// TwinCAT 3 PLC project lcls_plc_dream_vac
// ProgramVersion: 3.1.4022.7
// libraries:
//   LCLS General, * (SLAC)
//   LCLS Vacuum, * (SLAC - LCLS)
//   LCLSVacuumSerialDriverLib, * (SLAC - LCLS)
//   PMPS, * (SLAC - LCLS)
//   Tc2_SerialCom, * (Beckhoff Automation GmbH)
//   Tc2_Standard, * (Beckhoff Automation GmbH)
//   Tc2_System, * (Beckhoff Automation GmbH)
//   Tc3_Module, * (Beckhoff Automation GmbH)
// project tree:
//   DUTs/ E_Op.TcDUT, E_OpStep.TcDUT
//   GVLs/ GVL_Automation.TcGVL, GVL_Constants.TcGVL, GVL_FWM.TcGVL, GVL_PLC_Interface.TcGVL, GVL_Serial_Com.TcGVL, GVL_TC.TcGVL, GVL_VAC_GAUGES.TcGVL, GVL_VAC_PUMPS.TcGVL, GVL_VAC_VALVES.TcGVL, GVL_Variables.TcGVL
//   / PlcTask.TcTTO, Serial_COM.TcTTO
//   POUs/Automation/Abstracts/ FB_Operation.TcPOU
//   POUs/Automation/ FB_VentMcCat.TcPOU, FB_AtVacuum.TcPOU
//   POUs/Functions/ F_AllPumpsRunning.TcPOU, F_IsValidStateTransition.TcPOU, F_PressAtVacSP.TcPOU, F_TurboIlkLogic.TcPOU
//   POUs/ PRG_AUTOMATION.TcPOU, MAIN.TcPOU, PRG_COM.TcPOU, PRG_ECAT_CHECK.TcPOU, PRG_GAUGES.TcPOU, PRG_HV_ILK.TcPOU, PRG_COIL_PS_ILK.TcPOU, PRG_TC.TcPOU, PRG_TURBO_PUMPS.TcPOU, PRG_VALVES.TcPOU
// real-time tasks:
//   TASK PlcTask: cycle T#10ms, priority 20, ADS port 350
//   TASK Serial_COM: cycle T#2ms, priority 19, ADS port 351
// I/O:
//   DEVICE Device 1 (EtherCAT), AmsNetId 172.21.132.159.2.1
//     R20_DRL_03_CX0_EK1200 [EK1200-5000 EtherCAT Power supply (2A E-Bus)]
//       R20_DRL_03_E1_EL2202
//       R20_DRL_03_E2_EL6070 [EL6070 1Ch. Licensing-Terminal]
//       R20_DRL_03_E3_EL9070 [EL9070 Shield terminal]
//       R20_DRL_03_E4_EL1004 [EL1004 4Ch. Dig. Input 24V, 3ms]
//       R20_DRL_03_E5_EL1004 [EL1004 4Ch. Dig. Input 24V, 3ms]
//       R20_DRL_03_E6_EL1004
//       R20_DRL_03_E7_EL2794 [EL2794 4Ch. Dig. Output 24V AC/DC, 2A, short-circuit-proof]
//       R20_DRL_03_E8_EL2794 [EL2794 4Ch. Dig. Output 24V AC/DC, 2A, short-circuit-proof]
//       R20_DRL_03_E9_EL6001 [EL6001 Interface (RS232)]
//       R20_DRL_03_E10_EL6001 [EL6001 Interface (RS232)]
//       R20_DRL_03_E11_EL6001 [EL6001 Interface (RS232)]
//       R20_DRL_03_E12_EL6001 [EL6001 Interface (RS232)]
//       R20_DRL_03_E13_EL9505 [EL9505 Power supply terminal 5V]
//       R20_DRL_03_E14_EL6695 [EL6695 EtherCAT Bridge terminal (Primary)]
//       R20_DRL_03_E15_EL1122 [EK1122 2 port EtherCAT junction]
//         K4S8_DRL_03_EK0_EK1100 [EK1100 EtherCAT Coupler (2A E-Bus)]
//           K4S8_DRL_03_E1_EL2624 [EL2624 4Ch. Relay Output, NO (125V AC / 30V DC)]
//           K4S8_DRL_03_E2_EL9184 [EL9184 Potential Connection, 8 x 24V, 8 x Ground]
//           K4S8_DRL_03_E3_EL9070 [EL9070 Shield terminal]
//           K4S8_DRL_03_E4_EL1084 [EL1084 4Ch. Dig. Input 24V, 3ms, negative]
//           K4S8_DRL_03_E5_EL3174-0002 [EL3174-0002 4Ch. Ana. Input +/-10V, +/-20mA 16 Bit, Isolated Channels]
//           K4S8_DRL_03_E6_EL3174-0002 [EL3174-0002 4Ch. Ana. Input +/-10V, +/-20mA 16 Bit, Isolated Channels]
//           K4S8_DRL_03_E7_EL9505 [EL9505 Power supply terminal 5V]
//           K4S8_DRL_03_E8_EL1124 [EL1124 4Ch. Dig. Input 5V, 10µs, Sensor Power]
//           K4S8_DRL_03_E9_EL9410 [EL9410 E-Bus Power Supplier  (Diagnostics)]
//           K4S8_DRL_03_E10_EL1004 [EL1004 4Ch. Dig. Input 24V, 3ms]
//           K4S8_DRL_03_E11_EL2004 [EL2004 4Ch. Dig. Output 24V, 0.5A]
//           K4S8_DRL_03_E12_EL6021 [EL6021 Interface (RS422/485)]
//           K4S8_DRL_03_E13_EL1004 [EL1004 4Ch. Dig. Input 24V, 3ms]
//           K4S8_DRL_03_E14_EL2004 [EL2004 4Ch. Dig. Output 24V, 0.5A]
//           K4S8_DRL_03_E15_EL6021 [EL6021 Interface (RS422/485)]
//           K4S8_DRL_03_E16_EL1004 [EL1004 4Ch. Dig. Input 24V, 3ms]
//           K4S8_DRL_03_E17_EL2004 [EL2004 4Ch. Dig. Output 24V, 0.5A]
//           K4S8_DRL_03_E18_EL6021 [EL6021 Interface (RS422/485)]
//           K4S8_DRL_03_E19_EL1004 [EL1004 4Ch. Dig. Input 24V, 3ms]
//           K4S8_DRL_03_E20_EL2004 [EL2004 4Ch. Dig. Output 24V, 0.5A]
//           K4S8_DRL_03_E21_EL3052 [EL3052 2Ch. Ana. Input 4-20mA]
//           K4S8_DRL_03_E22_EL3314 [EL3314 4Ch. Ana. Input Thermocouple (TC)]
//           K4S8_DRL_03_E23_EL3314 [EL3314 4Ch. Ana. Input Thermocouple (TC)]
//           K4S8_DRL_03_E24_EL9011
//         K4S8_DRL_04_EK0_EK1100 [EK1100 EtherCAT Coupler (2A E-Bus)]
//           K4S8_DRL_04_E1_EL1004 [EL1004 4Ch. Dig. Input 24V, 3ms]
//           K4S8_DRL_04_E2_EL2004 [EL2004 4Ch. Dig. Output 24V, 0.5A]
//           K4S8_DRL_04_E3_EL1004 [EL1004 4Ch. Dig. Input 24V, 3ms]
//           K4S8_DRL_04_E4_EL1004 [EL1004 4Ch. Dig. Input 24V, 3ms]
//           K4S8_DRL_04_E5_EL2794 [EL2794 4Ch. Dig. Output 24V AC/DC, 2A, short-circuit-proof]
//           K4S8_DRL_04_E6_EL6001 [EL6001 Interface (RS232)]
//           K4S8_DRL_04_E7_EL6001 [EL6001 Interface (RS232)]
//           K4S8_DRL_04_E8_EL6001 [EL6001 Interface (RS232)]
//           K4S8_DRL_04_E9_EL1004 [EL1004 4Ch. Dig. Input 24V, 3ms]
//           K4S8_DRL_04_E10_EL1004 [EL1004 4Ch. Dig. Input 24V, 3ms]
//           K4S8_DRL_04_E11_EL2004
//           K4S8_DRL_04_E12_EL9184 [EL9184 Potential Connection, 8 x 24V, 8 x Ground]
//           K4S8_DRL_04_E13_EL9070 [EL9070 Shield terminal]
//           K4S8_DRL_04_E14_EL2624 [EL2624 4Ch. Relay Output, NO (125V AC / 30V DC)]
//           K4S8_DRL_04_E15_EL1084 [EL1084 4Ch. Dig. Input 24V, 3ms, negative]
//           K4S8_DRL_04_E16_EL3174-0002 [EL3174-0002 4Ch. Ana. Input +/-10V, +/-20mA 16 Bit, Isolated Channels]
//           K4S8_DRL_04_E17_EL6001 [EL6001 Interface (RS232)]
//           K4S8_DRL_04_E18_EL9011
//         K4S8_DRL_04_EP1_EP4374-0002 [EP4374-0002 2Ch. Ana. Input +/-10V, 0-10V, 0/4-20mA configurable; 2Ch. Ana. Output +/-10V, 0-10V, 0/4-20mA configurable]
//         K4S8_DRL_04_EP2_EP4374-0002 [EP4374-0002 2Ch. Ana. Input +/-10V, 0-10V, 0/4-20mA configurable; 2Ch. Ana. Output +/-10V, 0-10V, 0/4-20mA configurable]
//         R03_DRL_01_EK1100 [EK1100 EtherCAT Coupler (2A E-Bus)]
//           R03_DRL_01_E1_EL1004 [EL1004 4Ch. Dig. Input 24V, 3ms]
//           R03_DRL_01_E2_EL2624 [EL2624 4Ch. Relay Output, NO (125V AC / 30V DC)]
//           R03_DRL_01_E3_EL3174-0002 [EL3174-0002 4Ch. Ana. Input +/-10V, +/-20mA 16 Bit, Isolated Channels]
//           R03_DRL_01_E4_EK1110 [EK1110 EtherCAT extension]
//         WALL_E_PPL_01_EP1_EP4374-0002 [EP4374-0002 2Ch. Ana. Input +/-10V, 0-10V, 0/4-20mA configurable; 2Ch. Ana. Output +/-10V, 0-10V, 0/4-20mA configurable]
//         WALL_E_PPL_01_EP2_EP2338-0002 [EP2338-0002 8 Ch. Dig. Input/Output 24V, 0,5A, M12]
// variable links:
//   lcls_plc_dream_vac Instance <-> Device 1 (EtherCAT)/R20_DRL_03_CX0_EK1200/R20_DRL_03_E10_EL6001
//     Serial_COM Inputs/GVL_Serial_Com.stComIn_DREAM_DP3_PTM_01/D[0] <-> COM Inputs/Data In 0
//     Serial_COM Inputs/GVL_Serial_Com.stComIn_DREAM_DP3_PTM_01/D[10] <-> COM Inputs/Data In 10
//     Serial_COM Inputs/GVL_Serial_Com.stComIn_DREAM_DP3_PTM_01/D[11] <-> COM Inputs/Data In 11
//     Serial_COM Inputs/GVL_Serial_Com.stComIn_DREAM_DP3_PTM_01/D[12] <-> COM Inputs/Data In 12
//     Serial_COM Inputs/GVL_Serial_Com.stComIn_DREAM_DP3_PTM_01/D[13] <-> COM Inputs/Data In 13
//     Serial_COM Inputs/GVL_Serial_Com.stComIn_DREAM_DP3_PTM_01/D[14] <-> COM Inputs/Data In 14
//     Serial_COM Inputs/GVL_Serial_Com.stComIn_DREAM_DP3_PTM_01/D[15] <-> COM Inputs/Data In 15
//     Serial_COM Inputs/GVL_Serial_Com.stComIn_DREAM_DP3_PTM_01/D[16] <-> COM Inputs/Data In 16
//     Serial_COM Inputs/GVL_Serial_Com.stComIn_DREAM_DP3_PTM_01/D[17] <-> COM Inputs/Data In 17
//     Serial_COM Inputs/GVL_Serial_Com.stComIn_DREAM_DP3_PTM_01/D[18] <-> COM Inputs/Data In 18
//     Serial_COM Inputs/GVL_Serial_Com.stComIn_DREAM_DP3_PTM_01/D[19] <-> COM Inputs/Data In 19
//     Serial_COM Inputs/GVL_Serial_Com.stComIn_DREAM_DP3_PTM_01/D[1] <-> COM Inputs/Data In 1
//     Serial_COM Inputs/GVL_Serial_Com.stComIn_DREAM_DP3_PTM_01/D[20] <-> COM Inputs/Data In 20
//     Serial_COM Inputs/GVL_Serial_Com.stComIn_DREAM_DP3_PTM_01/D[21] <-> COM Inputs/Data In 21
//     Serial_COM Inputs/GVL_Serial_Com.stComIn_DREAM_DP3_PTM_01/D[2] <-> COM Inputs/Data In 2
//     Serial_COM Inputs/GVL_Serial_Com.stComIn_DREAM_DP3_PTM_01/D[3] <-> COM Inputs/Data In 3
//     Serial_COM Inputs/GVL_Serial_Com.stComIn_DREAM_DP3_PTM_01/D[4] <-> COM Inputs/Data In 4
//     Serial_COM Inputs/GVL_Serial_Com.stComIn_DREAM_DP3_PTM_01/D[5] <-> COM Inputs/Data In 5
//     Serial_COM Inputs/GVL_Serial_Com.stComIn_DREAM_DP3_PTM_01/D[6] <-> COM Inputs/Data In 6
//     Serial_COM Inputs/GVL_Serial_Com.stComIn_DREAM_DP3_PTM_01/D[7] <-> COM Inputs/Data In 7
//     Serial_COM Inputs/GVL_Serial_Com.stComIn_DREAM_DP3_PTM_01/D[8] <-> COM Inputs/Data In 8
//     Serial_COM Inputs/GVL_Serial_Com.stComIn_DREAM_DP3_PTM_01/D[9] <-> COM Inputs/Data In 9
//     Serial_COM Inputs/GVL_Serial_Com.stComIn_DREAM_DP3_PTM_01/Status <-> COM Inputs/Status
//     Serial_COM Outputs/GVL_Serial_Com.stComOut_DREAM_DP3_PTM_01/Ctrl <-> COM Outputs/Ctrl
//     Serial_COM Outputs/GVL_Serial_Com.stComOut_DREAM_DP3_PTM_01/D[0] <-> COM Outputs/Data Out 0
//     Serial_COM Outputs/GVL_Serial_Com.stComOut_DREAM_DP3_PTM_01/D[10] <-> COM Outputs/Data Out 10
//     Serial_COM Outputs/GVL_Serial_Com.stComOut_DREAM_DP3_PTM_01/D[11] <-> COM Outputs/Data Out 11
//     Serial_COM Outputs/GVL_Serial_Com.stComOut_DREAM_DP3_PTM_01/D[12] <-> COM Outputs/Data Out 12
//     Serial_COM Outputs/GVL_Serial_Com.stComOut_DREAM_DP3_PTM_01/D[13] <-> COM Outputs/Data Out 13
//     Serial_COM Outputs/GVL_Serial_Com.stComOut_DREAM_DP3_PTM_01/D[14] <-> COM Outputs/Data Out 14
//     Serial_COM Outputs/GVL_Serial_Com.stComOut_DREAM_DP3_PTM_01/D[15] <-> COM Outputs/Data Out 15
//     Serial_COM Outputs/GVL_Serial_Com.stComOut_DREAM_DP3_PTM_01/D[16] <-> COM Outputs/Data Out 16
//     Serial_COM Outputs/GVL_Serial_Com.stComOut_DREAM_DP3_PTM_01/D[17] <-> COM Outputs/Data Out 17
//     Serial_COM Outputs/GVL_Serial_Com.stComOut_DREAM_DP3_PTM_01/D[18] <-> COM Outputs/Data Out 18
//     Serial_COM Outputs/GVL_Serial_Com.stComOut_DREAM_DP3_PTM_01/D[19] <-> COM Outputs/Data Out 19
//     Serial_COM Outputs/GVL_Serial_Com.stComOut_DREAM_DP3_PTM_01/D[1] <-> COM Outputs/Data Out 1
//     Serial_COM Outputs/GVL_Serial_Com.stComOut_DREAM_DP3_PTM_01/D[20] <-> COM Outputs/Data Out 20
//     Serial_COM Outputs/GVL_Serial_Com.stComOut_DREAM_DP3_PTM_01/D[21] <-> COM Outputs/Data Out 21
//     Serial_COM Outputs/GVL_Serial_Com.stComOut_DREAM_DP3_PTM_01/D[2] <-> COM Outputs/Data Out 2
//     Serial_COM Outputs/GVL_Serial_Com.stComOut_DREAM_DP3_PTM_01/D[3] <-> COM Outputs/Data Out 3
//     Serial_COM Outputs/GVL_Serial_Com.stComOut_DREAM_DP3_PTM_01/D[4] <-> COM Outputs/Data Out 4
//     Serial_COM Outputs/GVL_Serial_Com.stComOut_DREAM_DP3_PTM_01/D[5] <-> COM Outputs/Data Out 5
//     Serial_COM Outputs/GVL_Serial_Com.stComOut_DREAM_DP3_PTM_01/D[6] <-> COM Outputs/Data Out 6
//     Serial_COM Outputs/GVL_Serial_Com.stComOut_DREAM_DP3_PTM_01/D[7] <-> COM Outputs/Data Out 7
//     Serial_COM Outputs/GVL_Serial_Com.stComOut_DREAM_DP3_PTM_01/D[8] <-> COM Outputs/Data Out 8
//     Serial_COM Outputs/GVL_Serial_Com.stComOut_DREAM_DP3_PTM_01/D[9] <-> COM Outputs/Data Out 9
//   lcls_plc_dream_vac Instance <-> Device 1 (EtherCAT)/R20_DRL_03_CX0_EK1200/R20_DRL_03_E11_EL6001
//     Serial_COM Inputs/GVL_Serial_Com.stComIn_DREAM_MC_PTM_01/D[0] <-> COM Inputs/Data In 0
//     Serial_COM Inputs/GVL_Serial_Com.stComIn_DREAM_MC_PTM_01/D[10] <-> COM Inputs/Data In 10
//     Serial_COM Inputs/GVL_Serial_Com.stComIn_DREAM_MC_PTM_01/D[11] <-> COM Inputs/Data In 11
//     Serial_COM Inputs/GVL_Serial_Com.stComIn_DREAM_MC_PTM_01/D[12] <-> COM Inputs/Data In 12
//     Serial_COM Inputs/GVL_Serial_Com.stComIn_DREAM_MC_PTM_01/D[13] <-> COM Inputs/Data In 13
//     Serial_COM Inputs/GVL_Serial_Com.stComIn_DREAM_MC_PTM_01/D[14] <-> COM Inputs/Data In 14
//     Serial_COM Inputs/GVL_Serial_Com.stComIn_DREAM_MC_PTM_01/D[15] <-> COM Inputs/Data In 15
//     Serial_COM Inputs/GVL_Serial_Com.stComIn_DREAM_MC_PTM_01/D[16] <-> COM Inputs/Data In 16
//     Serial_COM Inputs/GVL_Serial_Com.stComIn_DREAM_MC_PTM_01/D[17] <-> COM Inputs/Data In 17
//     Serial_COM Inputs/GVL_Serial_Com.stComIn_DREAM_MC_PTM_01/D[18] <-> COM Inputs/Data In 18
//     Serial_COM Inputs/GVL_Serial_Com.stComIn_DREAM_MC_PTM_01/D[19] <-> COM Inputs/Data In 19
//     Serial_COM Inputs/GVL_Serial_Com.stComIn_DREAM_MC_PTM_01/D[1] <-> COM Inputs/Data In 1
//     Serial_COM Inputs/GVL_Serial_Com.stComIn_DREAM_MC_PTM_01/D[20] <-> COM Inputs/Data In 20
//     Serial_COM Inputs/GVL_Serial_Com.stComIn_DREAM_MC_PTM_01/D[21] <-> COM Inputs/Data In 21
//     Serial_COM Inputs/GVL_Serial_Com.stComIn_DREAM_MC_PTM_01/D[2] <-> COM Inputs/Data In 2
//     Serial_COM Inputs/GVL_Serial_Com.stComIn_DREAM_MC_PTM_01/D[3] <-> COM Inputs/Data In 3
//     Serial_COM Inputs/GVL_Serial_Com.stComIn_DREAM_MC_PTM_01/D[4] <-> COM Inputs/Data In 4
//     Serial_COM Inputs/GVL_Serial_Com.stComIn_DREAM_MC_PTM_01/D[5] <-> COM Inputs/Data In 5
//     Serial_COM Inputs/GVL_Serial_Com.stComIn_DREAM_MC_PTM_01/D[6] <-> COM Inputs/Data In 6
//     Serial_COM Inputs/GVL_Serial_Com.stComIn_DREAM_MC_PTM_01/D[7] <-> COM Inputs/Data In 7
//     Serial_COM Inputs/GVL_Serial_Com.stComIn_DREAM_MC_PTM_01/D[8] <-> COM Inputs/Data In 8
//     Serial_COM Inputs/GVL_Serial_Com.stComIn_DREAM_MC_PTM_01/D[9] <-> COM Inputs/Data In 9
//     Serial_COM Inputs/GVL_Serial_Com.stComIn_DREAM_MC_PTM_01/Status <-> COM Inputs/Status
//     Serial_COM Outputs/GVL_Serial_Com.stComOut_DREAM_MC_PTM_01/Ctrl <-> COM Outputs/Ctrl
//     Serial_COM Outputs/GVL_Serial_Com.stComOut_DREAM_MC_PTM_01/D[0] <-> COM Outputs/Data Out 0
//     Serial_COM Outputs/GVL_Serial_Com.stComOut_DREAM_MC_PTM_01/D[10] <-> COM Outputs/Data Out 10
//     Serial_COM Outputs/GVL_Serial_Com.stComOut_DREAM_MC_PTM_01/D[11] <-> COM Outputs/Data Out 11
//     Serial_COM Outputs/GVL_Serial_Com.stComOut_DREAM_MC_PTM_01/D[12] <-> COM Outputs/Data Out 12
//     Serial_COM Outputs/GVL_Serial_Com.stComOut_DREAM_MC_PTM_01/D[13] <-> COM Outputs/Data Out 13
//     Serial_COM Outputs/GVL_Serial_Com.stComOut_DREAM_MC_PTM_01/D[14] <-> COM Outputs/Data Out 14
//     Serial_COM Outputs/GVL_Serial_Com.stComOut_DREAM_MC_PTM_01/D[15] <-> COM Outputs/Data Out 15
//     Serial_COM Outputs/GVL_Serial_Com.stComOut_DREAM_MC_PTM_01/D[16] <-> COM Outputs/Data Out 16
//     Serial_COM Outputs/GVL_Serial_Com.stComOut_DREAM_MC_PTM_01/D[17] <-> COM Outputs/Data Out 17
//     Serial_COM Outputs/GVL_Serial_Com.stComOut_DREAM_MC_PTM_01/D[18] <-> COM Outputs/Data Out 18
//     Serial_COM Outputs/GVL_Serial_Com.stComOut_DREAM_MC_PTM_01/D[19] <-> COM Outputs/Data Out 19
//     Serial_COM Outputs/GVL_Serial_Com.stComOut_DREAM_MC_PTM_01/D[1] <-> COM Outputs/Data Out 1
//     Serial_COM Outputs/GVL_Serial_Com.stComOut_DREAM_MC_PTM_01/D[20] <-> COM Outputs/Data Out 20
//     Serial_COM Outputs/GVL_Serial_Com.stComOut_DREAM_MC_PTM_01/D[21] <-> COM Outputs/Data Out 21
//     Serial_COM Outputs/GVL_Serial_Com.stComOut_DREAM_MC_PTM_01/D[2] <-> COM Outputs/Data Out 2
//     Serial_COM Outputs/GVL_Serial_Com.stComOut_DREAM_MC_PTM_01/D[3] <-> COM Outputs/Data Out 3
//     Serial_COM Outputs/GVL_Serial_Com.stComOut_DREAM_MC_PTM_01/D[4] <-> COM Outputs/Data Out 4
//     Serial_COM Outputs/GVL_Serial_Com.stComOut_DREAM_MC_PTM_01/D[5] <-> COM Outputs/Data Out 5
//     Serial_COM Outputs/GVL_Serial_Com.stComOut_DREAM_MC_PTM_01/D[6] <-> COM Outputs/Data Out 6
//     Serial_COM Outputs/GVL_Serial_Com.stComOut_DREAM_MC_PTM_01/D[7] <-> COM Outputs/Data Out 7
//     Serial_COM Outputs/GVL_Serial_Com.stComOut_DREAM_MC_PTM_01/D[8] <-> COM Outputs/Data Out 8
//     Serial_COM Outputs/GVL_Serial_Com.stComOut_DREAM_MC_PTM_01/D[9] <-> COM Outputs/Data Out 9
//   lcls_plc_dream_vac Instance <-> Device 1 (EtherCAT)/R20_DRL_03_CX0_EK1200/R20_DRL_03_E12_EL6001
//     Serial_COM Inputs/GVL_Serial_Com.stComIn_DREAM_MC_PTM_02/D[0] <-> COM Inputs/Data In 0
//     Serial_COM Inputs/GVL_Serial_Com.stComIn_DREAM_MC_PTM_02/D[10] <-> COM Inputs/Data In 10
//     Serial_COM Inputs/GVL_Serial_Com.stComIn_DREAM_MC_PTM_02/D[11] <-> COM Inputs/Data In 11
//     Serial_COM Inputs/GVL_Serial_Com.stComIn_DREAM_MC_PTM_02/D[12] <-> COM Inputs/Data In 12
//     Serial_COM Inputs/GVL_Serial_Com.stComIn_DREAM_MC_PTM_02/D[13] <-> COM Inputs/Data In 13
//     Serial_COM Inputs/GVL_Serial_Com.stComIn_DREAM_MC_PTM_02/D[14] <-> COM Inputs/Data In 14
//     Serial_COM Inputs/GVL_Serial_Com.stComIn_DREAM_MC_PTM_02/D[15] <-> COM Inputs/Data In 15
//     Serial_COM Inputs/GVL_Serial_Com.stComIn_DREAM_MC_PTM_02/D[16] <-> COM Inputs/Data In 16
//     Serial_COM Inputs/GVL_Serial_Com.stComIn_DREAM_MC_PTM_02/D[17] <-> COM Inputs/Data In 17
//     Serial_COM Inputs/GVL_Serial_Com.stComIn_DREAM_MC_PTM_02/D[18] <-> COM Inputs/Data In 18
//     Serial_COM Inputs/GVL_Serial_Com.stComIn_DREAM_MC_PTM_02/D[19] <-> COM Inputs/Data In 19
//     Serial_COM Inputs/GVL_Serial_Com.stComIn_DREAM_MC_PTM_02/D[1] <-> COM Inputs/Data In 1
//     Serial_COM Inputs/GVL_Serial_Com.stComIn_DREAM_MC_PTM_02/D[20] <-> COM Inputs/Data In 20
//     Serial_COM Inputs/GVL_Serial_Com.stComIn_DREAM_MC_PTM_02/D[21] <-> COM Inputs/Data In 21
//     Serial_COM Inputs/GVL_Serial_Com.stComIn_DREAM_MC_PTM_02/D[2] <-> COM Inputs/Data In 2
//     Serial_COM Inputs/GVL_Serial_Com.stComIn_DREAM_MC_PTM_02/D[3] <-> COM Inputs/Data In 3
//     Serial_COM Inputs/GVL_Serial_Com.stComIn_DREAM_MC_PTM_02/D[4] <-> COM Inputs/Data In 4
//     Serial_COM Inputs/GVL_Serial_Com.stComIn_DREAM_MC_PTM_02/D[5] <-> COM Inputs/Data In 5
//     Serial_COM Inputs/GVL_Serial_Com.stComIn_DREAM_MC_PTM_02/D[6] <-> COM Inputs/Data In 6
//     Serial_COM Inputs/GVL_Serial_Com.stComIn_DREAM_MC_PTM_02/D[7] <-> COM Inputs/Data In 7
//     Serial_COM Inputs/GVL_Serial_Com.stComIn_DREAM_MC_PTM_02/D[8] <-> COM Inputs/Data In 8
//     Serial_COM Inputs/GVL_Serial_Com.stComIn_DREAM_MC_PTM_02/D[9] <-> COM Inputs/Data In 9
//     Serial_COM Inputs/GVL_Serial_Com.stComIn_DREAM_MC_PTM_02/Status <-> COM Inputs/Status
//     Serial_COM Outputs/GVL_Serial_Com.stComOut_DREAM_MC_PTM_02/Ctrl <-> COM Outputs/Ctrl
//     Serial_COM Outputs/GVL_Serial_Com.stComOut_DREAM_MC_PTM_02/D[0] <-> COM Outputs/Data Out 0
//     Serial_COM Outputs/GVL_Serial_Com.stComOut_DREAM_MC_PTM_02/D[10] <-> COM Outputs/Data Out 10
//     Serial_COM Outputs/GVL_Serial_Com.stComOut_DREAM_MC_PTM_02/D[11] <-> COM Outputs/Data Out 11
//     Serial_COM Outputs/GVL_Serial_Com.stComOut_DREAM_MC_PTM_02/D[12] <-> COM Outputs/Data Out 12
//     Serial_COM Outputs/GVL_Serial_Com.stComOut_DREAM_MC_PTM_02/D[13] <-> COM Outputs/Data Out 13
//     Serial_COM Outputs/GVL_Serial_Com.stComOut_DREAM_MC_PTM_02/D[14] <-> COM Outputs/Data Out 14
//     Serial_COM Outputs/GVL_Serial_Com.stComOut_DREAM_MC_PTM_02/D[15] <-> COM Outputs/Data Out 15
//     Serial_COM Outputs/GVL_Serial_Com.stComOut_DREAM_MC_PTM_02/D[16] <-> COM Outputs/Data Out 16
//     Serial_COM Outputs/GVL_Serial_Com.stComOut_DREAM_MC_PTM_02/D[17] <-> COM Outputs/Data Out 17
//     Serial_COM Outputs/GVL_Serial_Com.stComOut_DREAM_MC_PTM_02/D[18] <-> COM Outputs/Data Out 18
//     Serial_COM Outputs/GVL_Serial_Com.stComOut_DREAM_MC_PTM_02/D[19] <-> COM Outputs/Data Out 19
//     Serial_COM Outputs/GVL_Serial_Com.stComOut_DREAM_MC_PTM_02/D[1] <-> COM Outputs/Data Out 1
//     Serial_COM Outputs/GVL_Serial_Com.stComOut_DREAM_MC_PTM_02/D[20] <-> COM Outputs/Data Out 20
//     Serial_COM Outputs/GVL_Serial_Com.stComOut_DREAM_MC_PTM_02/D[21] <-> COM Outputs/Data Out 21
//     Serial_COM Outputs/GVL_Serial_Com.stComOut_DREAM_MC_PTM_02/D[2] <-> COM Outputs/Data Out 2
//     Serial_COM Outputs/GVL_Serial_Com.stComOut_DREAM_MC_PTM_02/D[3] <-> COM Outputs/Data Out 3
//     Serial_COM Outputs/GVL_Serial_Com.stComOut_DREAM_MC_PTM_02/D[4] <-> COM Outputs/Data Out 4
//     Serial_COM Outputs/GVL_Serial_Com.stComOut_DREAM_MC_PTM_02/D[5] <-> COM Outputs/Data Out 5
//     Serial_COM Outputs/GVL_Serial_Com.stComOut_DREAM_MC_PTM_02/D[6] <-> COM Outputs/Data Out 6
//     Serial_COM Outputs/GVL_Serial_Com.stComOut_DREAM_MC_PTM_02/D[7] <-> COM Outputs/Data Out 7
//     Serial_COM Outputs/GVL_Serial_Com.stComOut_DREAM_MC_PTM_02/D[8] <-> COM Outputs/Data Out 8
//     Serial_COM Outputs/GVL_Serial_Com.stComOut_DREAM_MC_PTM_02/D[9] <-> COM Outputs/Data Out 9
//   lcls_plc_dream_vac Instance <-> Device 1 (EtherCAT)/R20_DRL_03_CX0_EK1200/R20_DRL_03_E14_EL6695
//     PlcTask Inputs/GVL_PLC_Interface.bEcatBridge_External_device_not_connected <-> SYNC Inputs/External device not connected
//     PlcTask Inputs/GVL_PLC_Interface.bEcatBridge_TxPDO_state <-> SYNC Inputs/TxPDO state
//     PlcTask Inputs/GVL_PLC_Interface.bEcatBridge_WcState <-> WcState/WcStateIn
//     PlcTask Inputs/GVL_PLC_Interface.bMotEcatBridge_External_device_not_connected <-> SYNC Inputs/External device not connected
//     PlcTask Inputs/GVL_PLC_Interface.bTMO_MR5K4_VWC_CLOSED_LS <-> IO Inputs/TMO_MR5K4_VWC_CLOSED_LS
//     PlcTask Inputs/GVL_PLC_Interface.bTMO_MR5K4_VWC_OPEN_LS <-> IO Inputs/TMO_MR5K4_VWC_OPEN_LS
//     PlcTask Inputs/GVL_PLC_Interface.bTMO_TM2K4_VWC_CLOSED_LS <-> IO Inputs/TMO_TM2K4_VWC_CLOSED_LS
//     PlcTask Inputs/GVL_PLC_Interface.bTMO_TM2K4_VWC_OPEN_LS <-> IO Inputs/TMO_TM2K4_VWC_OPEN_LS
//     PlcTask Inputs/GVL_PLC_Interface.sHUTCH_PLC_NAME <-> IO Inputs/HUTCH_PLC_NAME
//     PlcTask Outputs/GVL_PLC_Interface.bCLOSE_TMO_MR5K4_VWC <-> IO Outputs/CLOSE_TMO_MR5K4_VWC
//     PlcTask Outputs/GVL_PLC_Interface.bCLOSE_TMO_TM2K4_VWC <-> IO Outputs/CLOSE_TMO_TM2K4_VWC
//     PlcTask Outputs/GVL_PLC_Interface.bDREAM_HV_SAFETY_ENABLE <-> IO Outputs/DREAM_HV_SAFETY_ENABLE
//     PlcTask Outputs/GVL_PLC_Interface.bDREAM_MAIN_xAT_VAC <-> IO Outputs/DREAM_MAIN_xAT_VAC
//     PlcTask Outputs/GVL_PLC_Interface.bDREAM_MAIN_xPRESS_OK <-> IO Outputs/DREAM_MAIN_xPRESS_OK
//     PlcTask Outputs/GVL_PLC_Interface.bDREAM_TURBOS_ALL_AtSpd <-> IO Outputs/DREAM_TURBOS_ALL_AtSpd
//     PlcTask Outputs/GVL_PLC_Interface.fDREAM_MAIN_rPRESS <-> IO Outputs/DREAM_MAIN_rPRESS
//     PlcTask Outputs/GVL_PLC_Interface.sENDSTATION_PLC_NAME <-> IO Outputs/ENDSTATION_PLC_NAME
//   lcls_plc_dream_vac Instance <-> Device 1 (EtherCAT)/R20_DRL_03_CX0_EK1200/R20_DRL_03_E15_EL1122/K4S8_DRL_03_EK0_EK1100/K4S8_DRL_03_E10_EL1004
//     PlcTask Inputs/GVL_VAC_VALVES.DREAM_DP1_VRC_01.i_xClsLS <-> Channel 2/Input
//     PlcTask Inputs/GVL_VAC_VALVES.DREAM_DP1_VRC_02.i_xClsLS <-> Channel 4/Input
//     PlcTask Inputs/GVL_VAC_VALVES.DREAM_DP1_VRC_01.i_xOpnLS <-> Channel 1/Input
//     PlcTask Inputs/GVL_VAC_VALVES.DREAM_DP1_VRC_02.i_xOpnLS <-> Channel 3/Input
//   lcls_plc_dream_vac Instance <-> Device 1 (EtherCAT)/R20_DRL_03_CX0_EK1200/R20_DRL_03_E15_EL1122/K4S8_DRL_03_EK0_EK1100/K4S8_DRL_03_E11_EL2004
//     PlcTask Outputs/GVL_VAC_VALVES.DREAM_DP1_VRC_01.q_xOPN_DO <-> Channel 2/Output
//     PlcTask Outputs/GVL_VAC_VALVES.DREAM_DP1_VRC_02.q_xCLS_DO <-> Channel 1/Output
//   lcls_plc_dream_vac Instance <-> Device 1 (EtherCAT)/R20_DRL_03_CX0_EK1200/R20_DRL_03_E15_EL1122/K4S8_DRL_03_EK0_EK1100/K4S8_DRL_03_E12_EL6021
//     Serial_COM Inputs/GVL_Serial_Com.stComIn_DREAM_NC_PTM_01/D[0] <-> COM TxPDO-Map Inputs/Data In 0
//     Serial_COM Inputs/GVL_Serial_Com.stComIn_DREAM_NC_PTM_01/D[10] <-> COM TxPDO-Map Inputs/Data In 10
//     Serial_COM Inputs/GVL_Serial_Com.stComIn_DREAM_NC_PTM_01/D[11] <-> COM TxPDO-Map Inputs/Data In 11
//     Serial_COM Inputs/GVL_Serial_Com.stComIn_DREAM_NC_PTM_01/D[12] <-> COM TxPDO-Map Inputs/Data In 12
//     Serial_COM Inputs/GVL_Serial_Com.stComIn_DREAM_NC_PTM_01/D[13] <-> COM TxPDO-Map Inputs/Data In 13
//     Serial_COM Inputs/GVL_Serial_Com.stComIn_DREAM_NC_PTM_01/D[14] <-> COM TxPDO-Map Inputs/Data In 14
//     Serial_COM Inputs/GVL_Serial_Com.stComIn_DREAM_NC_PTM_01/D[15] <-> COM TxPDO-Map Inputs/Data In 15
//     Serial_COM Inputs/GVL_Serial_Com.stComIn_DREAM_NC_PTM_01/D[16] <-> COM TxPDO-Map Inputs/Data In 16
//     Serial_COM Inputs/GVL_Serial_Com.stComIn_DREAM_NC_PTM_01/D[17] <-> COM TxPDO-Map Inputs/Data In 17
//     Serial_COM Inputs/GVL_Serial_Com.stComIn_DREAM_NC_PTM_01/D[18] <-> COM TxPDO-Map Inputs/Data In 18
//     Serial_COM Inputs/GVL_Serial_Com.stComIn_DREAM_NC_PTM_01/D[19] <-> COM TxPDO-Map Inputs/Data In 19
//     Serial_COM Inputs/GVL_Serial_Com.stComIn_DREAM_NC_PTM_01/D[1] <-> COM TxPDO-Map Inputs/Data In 1
//     Serial_COM Inputs/GVL_Serial_Com.stComIn_DREAM_NC_PTM_01/D[20] <-> COM TxPDO-Map Inputs/Data In 20
//     Serial_COM Inputs/GVL_Serial_Com.stComIn_DREAM_NC_PTM_01/D[21] <-> COM TxPDO-Map Inputs/Data In 21
//     Serial_COM Inputs/GVL_Serial_Com.stComIn_DREAM_NC_PTM_01/D[2] <-> COM TxPDO-Map Inputs/Data In 2
//     Serial_COM Inputs/GVL_Serial_Com.stComIn_DREAM_NC_PTM_01/D[3] <-> COM TxPDO-Map Inputs/Data In 3
//     Serial_COM Inputs/GVL_Serial_Com.stComIn_DREAM_NC_PTM_01/D[4] <-> COM TxPDO-Map Inputs/Data In 4
//     Serial_COM Inputs/GVL_Serial_Com.stComIn_DREAM_NC_PTM_01/D[5] <-> COM TxPDO-Map Inputs/Data In 5
//     Serial_COM Inputs/GVL_Serial_Com.stComIn_DREAM_NC_PTM_01/D[6] <-> COM TxPDO-Map Inputs/Data In 6
//     Serial_COM Inputs/GVL_Serial_Com.stComIn_DREAM_NC_PTM_01/D[7] <-> COM TxPDO-Map Inputs/Data In 7
//     Serial_COM Inputs/GVL_Serial_Com.stComIn_DREAM_NC_PTM_01/D[8] <-> COM TxPDO-Map Inputs/Data In 8
//     Serial_COM Inputs/GVL_Serial_Com.stComIn_DREAM_NC_PTM_01/D[9] <-> COM TxPDO-Map Inputs/Data In 9
//     Serial_COM Inputs/GVL_Serial_Com.stComIn_DREAM_NC_PTM_01/Status <-> COM TxPDO-Map Inputs/Status
//     Serial_COM Outputs/GVL_Serial_Com.stComOut_DREAM_NC_PTM_01/Ctrl <-> COM RxPDO-Map Outputs/Ctrl
//     Serial_COM Outputs/GVL_Serial_Com.stComOut_DREAM_NC_PTM_01/D[0] <-> COM RxPDO-Map Outputs/Data Out 0
//     Serial_COM Outputs/GVL_Serial_Com.stComOut_DREAM_NC_PTM_01/D[10] <-> COM RxPDO-Map Outputs/Data Out 10
//     Serial_COM Outputs/GVL_Serial_Com.stComOut_DREAM_NC_PTM_01/D[11] <-> COM RxPDO-Map Outputs/Data Out 11
//     Serial_COM Outputs/GVL_Serial_Com.stComOut_DREAM_NC_PTM_01/D[12] <-> COM RxPDO-Map Outputs/Data Out 12
//     Serial_COM Outputs/GVL_Serial_Com.stComOut_DREAM_NC_PTM_01/D[13] <-> COM RxPDO-Map Outputs/Data Out 13
//     Serial_COM Outputs/GVL_Serial_Com.stComOut_DREAM_NC_PTM_01/D[14] <-> COM RxPDO-Map Outputs/Data Out 14
//     Serial_COM Outputs/GVL_Serial_Com.stComOut_DREAM_NC_PTM_01/D[15] <-> COM RxPDO-Map Outputs/Data Out 15
//     Serial_COM Outputs/GVL_Serial_Com.stComOut_DREAM_NC_PTM_01/D[16] <-> COM RxPDO-Map Outputs/Data Out 16
//     Serial_COM Outputs/GVL_Serial_Com.stComOut_DREAM_NC_PTM_01/D[17] <-> COM RxPDO-Map Outputs/Data Out 17
//     Serial_COM Outputs/GVL_Serial_Com.stComOut_DREAM_NC_PTM_01/D[18] <-> COM RxPDO-Map Outputs/Data Out 18
//     Serial_COM Outputs/GVL_Serial_Com.stComOut_DREAM_NC_PTM_01/D[19] <-> COM RxPDO-Map Outputs/Data Out 19
//     Serial_COM Outputs/GVL_Serial_Com.stComOut_DREAM_NC_PTM_01/D[1] <-> COM RxPDO-Map Outputs/Data Out 1
//     Serial_COM Outputs/GVL_Serial_Com.stComOut_DREAM_NC_PTM_01/D[20] <-> COM RxPDO-Map Outputs/Data Out 20
//     Serial_COM Outputs/GVL_Serial_Com.stComOut_DREAM_NC_PTM_01/D[21] <-> COM RxPDO-Map Outputs/Data Out 21
//     Serial_COM Outputs/GVL_Serial_Com.stComOut_DREAM_NC_PTM_01/D[2] <-> COM RxPDO-Map Outputs/Data Out 2
//     Serial_COM Outputs/GVL_Serial_Com.stComOut_DREAM_NC_PTM_01/D[3] <-> COM RxPDO-Map Outputs/Data Out 3
//     Serial_COM Outputs/GVL_Serial_Com.stComOut_DREAM_NC_PTM_01/D[4] <-> COM RxPDO-Map Outputs/Data Out 4
//     Serial_COM Outputs/GVL_Serial_Com.stComOut_DREAM_NC_PTM_01/D[5] <-> COM RxPDO-Map Outputs/Data Out 5
//     Serial_COM Outputs/GVL_Serial_Com.stComOut_DREAM_NC_PTM_01/D[6] <-> COM RxPDO-Map Outputs/Data Out 6
//     Serial_COM Outputs/GVL_Serial_Com.stComOut_DREAM_NC_PTM_01/D[7] <-> COM RxPDO-Map Outputs/Data Out 7
//     Serial_COM Outputs/GVL_Serial_Com.stComOut_DREAM_NC_PTM_01/D[8] <-> COM RxPDO-Map Outputs/Data Out 8
//     Serial_COM Outputs/GVL_Serial_Com.stComOut_DREAM_NC_PTM_01/D[9] <-> COM RxPDO-Map Outputs/Data Out 9
//   lcls_plc_dream_vac Instance <-> Device 1 (EtherCAT)/R20_DRL_03_CX0_EK1200/R20_DRL_03_E15_EL1122/K4S8_DRL_03_EK0_EK1100/K4S8_DRL_03_E13_EL1004
//     PlcTask Inputs/GVL_VAC_PUMPS.DREAM_NC_PTM_01.i_xAtSpd <-> Channel 1/Input
//     PlcTask Inputs/GVL_VAC_PUMPS.DREAM_NC_PTM_01.i_xFaultNC <-> Channel 3/Input
//     PlcTask Inputs/GVL_VAC_PUMPS.DREAM_NC_PTM_01.i_xRemote <-> Channel 2/Input
//   lcls_plc_dream_vac Instance <-> Device 1 (EtherCAT)/R20_DRL_03_CX0_EK1200/R20_DRL_03_E15_EL1122/K4S8_DRL_03_EK0_EK1100/K4S8_DRL_03_E14_EL2004
//     PlcTask Outputs/GVL_VAC_PUMPS.DREAM_NC_PTM_01.q_PumpingStation <-> Channel 3/Output
//     PlcTask Outputs/GVL_VAC_PUMPS.DREAM_NC_PTM_01.q_RunDO <-> Channel 1/Output
//     PlcTask Outputs/GVL_VAC_PUMPS.DREAM_NC_PTM_01.q_xRemote <-> Channel 2/Output
//   lcls_plc_dream_vac Instance <-> Device 1 (EtherCAT)/R20_DRL_03_CX0_EK1200/R20_DRL_03_E15_EL1122/K4S8_DRL_03_EK0_EK1100/K4S8_DRL_03_E15_EL6021
//     Serial_COM Inputs/GVL_Serial_Com.stComIn_DREAM_NC_PTM_02/D[0] <-> COM TxPDO-Map Inputs/Data In 0
//     Serial_COM Inputs/GVL_Serial_Com.stComIn_DREAM_NC_PTM_02/D[10] <-> COM TxPDO-Map Inputs/Data In 10
//     Serial_COM Inputs/GVL_Serial_Com.stComIn_DREAM_NC_PTM_02/D[11] <-> COM TxPDO-Map Inputs/Data In 11
//     Serial_COM Inputs/GVL_Serial_Com.stComIn_DREAM_NC_PTM_02/D[12] <-> COM TxPDO-Map Inputs/Data In 12
//     Serial_COM Inputs/GVL_Serial_Com.stComIn_DREAM_NC_PTM_02/D[13] <-> COM TxPDO-Map Inputs/Data In 13
//     Serial_COM Inputs/GVL_Serial_Com.stComIn_DREAM_NC_PTM_02/D[14] <-> COM TxPDO-Map Inputs/Data In 14
//     Serial_COM Inputs/GVL_Serial_Com.stComIn_DREAM_NC_PTM_02/D[15] <-> COM TxPDO-Map Inputs/Data In 15
//     Serial_COM Inputs/GVL_Serial_Com.stComIn_DREAM_NC_PTM_02/D[16] <-> COM TxPDO-Map Inputs/Data In 16
//     Serial_COM Inputs/GVL_Serial_Com.stComIn_DREAM_NC_PTM_02/D[17] <-> COM TxPDO-Map Inputs/Data In 17
//     Serial_COM Inputs/GVL_Serial_Com.stComIn_DREAM_NC_PTM_02/D[18] <-> COM TxPDO-Map Inputs/Data In 18
//     Serial_COM Inputs/GVL_Serial_Com.stComIn_DREAM_NC_PTM_02/D[19] <-> COM TxPDO-Map Inputs/Data In 19
//     Serial_COM Inputs/GVL_Serial_Com.stComIn_DREAM_NC_PTM_02/D[1] <-> COM TxPDO-Map Inputs/Data In 1
//     Serial_COM Inputs/GVL_Serial_Com.stComIn_DREAM_NC_PTM_02/D[20] <-> COM TxPDO-Map Inputs/Data In 20
//     Serial_COM Inputs/GVL_Serial_Com.stComIn_DREAM_NC_PTM_02/D[21] <-> COM TxPDO-Map Inputs/Data In 21
//     Serial_COM Inputs/GVL_Serial_Com.stComIn_DREAM_NC_PTM_02/D[2] <-> COM TxPDO-Map Inputs/Data In 2
//     Serial_COM Inputs/GVL_Serial_Com.stComIn_DREAM_NC_PTM_02/D[3] <-> COM TxPDO-Map Inputs/Data In 3
//     Serial_COM Inputs/GVL_Serial_Com.stComIn_DREAM_NC_PTM_02/D[4] <-> COM TxPDO-Map Inputs/Data In 4
//     Serial_COM Inputs/GVL_Serial_Com.stComIn_DREAM_NC_PTM_02/D[5] <-> COM TxPDO-Map Inputs/Data In 5
//     Serial_COM Inputs/GVL_Serial_Com.stComIn_DREAM_NC_PTM_02/D[6] <-> COM TxPDO-Map Inputs/Data In 6
//     Serial_COM Inputs/GVL_Serial_Com.stComIn_DREAM_NC_PTM_02/D[7] <-> COM TxPDO-Map Inputs/Data In 7
//     Serial_COM Inputs/GVL_Serial_Com.stComIn_DREAM_NC_PTM_02/D[8] <-> COM TxPDO-Map Inputs/Data In 8
//     Serial_COM Inputs/GVL_Serial_Com.stComIn_DREAM_NC_PTM_02/D[9] <-> COM TxPDO-Map Inputs/Data In 9
//     Serial_COM Inputs/GVL_Serial_Com.stComIn_DREAM_NC_PTM_02/Status <-> COM TxPDO-Map Inputs/Status
//     Serial_COM Outputs/GVL_Serial_Com.stComOut_DREAM_NC_PTM_02/Ctrl <-> COM RxPDO-Map Outputs/Ctrl
//     Serial_COM Outputs/GVL_Serial_Com.stComOut_DREAM_NC_PTM_02/D[0] <-> COM RxPDO-Map Outputs/Data Out 0
//     Serial_COM Outputs/GVL_Serial_Com.stComOut_DREAM_NC_PTM_02/D[10] <-> COM RxPDO-Map Outputs/Data Out 10
//     Serial_COM Outputs/GVL_Serial_Com.stComOut_DREAM_NC_PTM_02/D[11] <-> COM RxPDO-Map Outputs/Data Out 11
//     Serial_COM Outputs/GVL_Serial_Com.stComOut_DREAM_NC_PTM_02/D[12] <-> COM RxPDO-Map Outputs/Data Out 12
//     Serial_COM Outputs/GVL_Serial_Com.stComOut_DREAM_NC_PTM_02/D[13] <-> COM RxPDO-Map Outputs/Data Out 13
//     Serial_COM Outputs/GVL_Serial_Com.stComOut_DREAM_NC_PTM_02/D[14] <-> COM RxPDO-Map Outputs/Data Out 14
//     Serial_COM Outputs/GVL_Serial_Com.stComOut_DREAM_NC_PTM_02/D[15] <-> COM RxPDO-Map Outputs/Data Out 15
//     Serial_COM Outputs/GVL_Serial_Com.stComOut_DREAM_NC_PTM_02/D[16] <-> COM RxPDO-Map Outputs/Data Out 16
//     Serial_COM Outputs/GVL_Serial_Com.stComOut_DREAM_NC_PTM_02/D[17] <-> COM RxPDO-Map Outputs/Data Out 17
//     Serial_COM Outputs/GVL_Serial_Com.stComOut_DREAM_NC_PTM_02/D[18] <-> COM RxPDO-Map Outputs/Data Out 18
//     Serial_COM Outputs/GVL_Serial_Com.stComOut_DREAM_NC_PTM_02/D[19] <-> COM RxPDO-Map Outputs/Data Out 19
//     Serial_COM Outputs/GVL_Serial_Com.stComOut_DREAM_NC_PTM_02/D[1] <-> COM RxPDO-Map Outputs/Data Out 1
//     Serial_COM Outputs/GVL_Serial_Com.stComOut_DREAM_NC_PTM_02/D[20] <-> COM RxPDO-Map Outputs/Data Out 20
//     Serial_COM Outputs/GVL_Serial_Com.stComOut_DREAM_NC_PTM_02/D[21] <-> COM RxPDO-Map Outputs/Data Out 21
//     Serial_COM Outputs/GVL_Serial_Com.stComOut_DREAM_NC_PTM_02/D[2] <-> COM RxPDO-Map Outputs/Data Out 2
//     Serial_COM Outputs/GVL_Serial_Com.stComOut_DREAM_NC_PTM_02/D[3] <-> COM RxPDO-Map Outputs/Data Out 3
//     Serial_COM Outputs/GVL_Serial_Com.stComOut_DREAM_NC_PTM_02/D[4] <-> COM RxPDO-Map Outputs/Data Out 4
//     Serial_COM Outputs/GVL_Serial_Com.stComOut_DREAM_NC_PTM_02/D[5] <-> COM RxPDO-Map Outputs/Data Out 5
//     Serial_COM Outputs/GVL_Serial_Com.stComOut_DREAM_NC_PTM_02/D[6] <-> COM RxPDO-Map Outputs/Data Out 6
//     Serial_COM Outputs/GVL_Serial_Com.stComOut_DREAM_NC_PTM_02/D[7] <-> COM RxPDO-Map Outputs/Data Out 7
//     Serial_COM Outputs/GVL_Serial_Com.stComOut_DREAM_NC_PTM_02/D[8] <-> COM RxPDO-Map Outputs/Data Out 8
//     Serial_COM Outputs/GVL_Serial_Com.stComOut_DREAM_NC_PTM_02/D[9] <-> COM RxPDO-Map Outputs/Data Out 9
//   lcls_plc_dream_vac Instance <-> Device 1 (EtherCAT)/R20_DRL_03_CX0_EK1200/R20_DRL_03_E15_EL1122/K4S8_DRL_03_EK0_EK1100/K4S8_DRL_03_E16_EL1004
//     PlcTask Inputs/GVL_VAC_PUMPS.DREAM_NC_PTM_02.i_xAtSpd <-> Channel 1/Input
//     PlcTask Inputs/GVL_VAC_PUMPS.DREAM_NC_PTM_02.i_xFaultNC <-> Channel 3/Input
//     PlcTask Inputs/GVL_VAC_PUMPS.DREAM_NC_PTM_02.i_xRemote <-> Channel 2/Input
//   lcls_plc_dream_vac Instance <-> Device 1 (EtherCAT)/R20_DRL_03_CX0_EK1200/R20_DRL_03_E15_EL1122/K4S8_DRL_03_EK0_EK1100/K4S8_DRL_03_E17_EL2004
//     PlcTask Outputs/GVL_VAC_PUMPS.DREAM_NC_PTM_02.q_PumpingStation <-> Channel 3/Output
//     PlcTask Outputs/GVL_VAC_PUMPS.DREAM_NC_PTM_02.q_RunDO <-> Channel 1/Output
//     PlcTask Outputs/GVL_VAC_PUMPS.DREAM_NC_PTM_02.q_xRemote <-> Channel 2/Output
//   lcls_plc_dream_vac Instance <-> Device 1 (EtherCAT)/R20_DRL_03_CX0_EK1200/R20_DRL_03_E15_EL1122/K4S8_DRL_03_EK0_EK1100/K4S8_DRL_03_E18_EL6021
//     Serial_COM Inputs/GVL_Serial_Com.stComIn_DREAM_DP1_PTM_01/D[0] <-> COM TxPDO-Map Inputs/Data In 0
//     Serial_COM Inputs/GVL_Serial_Com.stComIn_DREAM_DP1_PTM_01/D[10] <-> COM TxPDO-Map Inputs/Data In 10
//     Serial_COM Inputs/GVL_Serial_Com.stComIn_DREAM_DP1_PTM_01/D[11] <-> COM TxPDO-Map Inputs/Data In 11
//     Serial_COM Inputs/GVL_Serial_Com.stComIn_DREAM_DP1_PTM_01/D[12] <-> COM TxPDO-Map Inputs/Data In 12
//     Serial_COM Inputs/GVL_Serial_Com.stComIn_DREAM_DP1_PTM_01/D[13] <-> COM TxPDO-Map Inputs/Data In 13
//     Serial_COM Inputs/GVL_Serial_Com.stComIn_DREAM_DP1_PTM_01/D[14] <-> COM TxPDO-Map Inputs/Data In 14
//     Serial_COM Inputs/GVL_Serial_Com.stComIn_DREAM_DP1_PTM_01/D[15] <-> COM TxPDO-Map Inputs/Data In 15
//     Serial_COM Inputs/GVL_Serial_Com.stComIn_DREAM_DP1_PTM_01/D[16] <-> COM TxPDO-Map Inputs/Data In 16
//     Serial_COM Inputs/GVL_Serial_Com.stComIn_DREAM_DP1_PTM_01/D[17] <-> COM TxPDO-Map Inputs/Data In 17
//     Serial_COM Inputs/GVL_Serial_Com.stComIn_DREAM_DP1_PTM_01/D[18] <-> COM TxPDO-Map Inputs/Data In 18
//     Serial_COM Inputs/GVL_Serial_Com.stComIn_DREAM_DP1_PTM_01/D[19] <-> COM TxPDO-Map Inputs/Data In 19
//     Serial_COM Inputs/GVL_Serial_Com.stComIn_DREAM_DP1_PTM_01/D[1] <-> COM TxPDO-Map Inputs/Data In 1
//     Serial_COM Inputs/GVL_Serial_Com.stComIn_DREAM_DP1_PTM_01/D[20] <-> COM TxPDO-Map Inputs/Data In 20
//     Serial_COM Inputs/GVL_Serial_Com.stComIn_DREAM_DP1_PTM_01/D[21] <-> COM TxPDO-Map Inputs/Data In 21
//     Serial_COM Inputs/GVL_Serial_Com.stComIn_DREAM_DP1_PTM_01/D[2] <-> COM TxPDO-Map Inputs/Data In 2
//     Serial_COM Inputs/GVL_Serial_Com.stComIn_DREAM_DP1_PTM_01/D[3] <-> COM TxPDO-Map Inputs/Data In 3
//     Serial_COM Inputs/GVL_Serial_Com.stComIn_DREAM_DP1_PTM_01/D[4] <-> COM TxPDO-Map Inputs/Data In 4
//     Serial_COM Inputs/GVL_Serial_Com.stComIn_DREAM_DP1_PTM_01/D[5] <-> COM TxPDO-Map Inputs/Data In 5
//     Serial_COM Inputs/GVL_Serial_Com.stComIn_DREAM_DP1_PTM_01/D[6] <-> COM TxPDO-Map Inputs/Data In 6
//     Serial_COM Inputs/GVL_Serial_Com.stComIn_DREAM_DP1_PTM_01/D[7] <-> COM TxPDO-Map Inputs/Data In 7
//     Serial_COM Inputs/GVL_Serial_Com.stComIn_DREAM_DP1_PTM_01/D[8] <-> COM TxPDO-Map Inputs/Data In 8
//     Serial_COM Inputs/GVL_Serial_Com.stComIn_DREAM_DP1_PTM_01/D[9] <-> COM TxPDO-Map Inputs/Data In 9
//     Serial_COM Inputs/GVL_Serial_Com.stComIn_DREAM_DP1_PTM_01/Status <-> COM TxPDO-Map Inputs/Status
//     Serial_COM Outputs/GVL_Serial_Com.stComOut_DREAM_DP1_PTM_01/Ctrl <-> COM RxPDO-Map Outputs/Ctrl
//     Serial_COM Outputs/GVL_Serial_Com.stComOut_DREAM_DP1_PTM_01/D[0] <-> COM RxPDO-Map Outputs/Data Out 0
//     Serial_COM Outputs/GVL_Serial_Com.stComOut_DREAM_DP1_PTM_01/D[10] <-> COM RxPDO-Map Outputs/Data Out 10
//     Serial_COM Outputs/GVL_Serial_Com.stComOut_DREAM_DP1_PTM_01/D[11] <-> COM RxPDO-Map Outputs/Data Out 11
//     Serial_COM Outputs/GVL_Serial_Com.stComOut_DREAM_DP1_PTM_01/D[12] <-> COM RxPDO-Map Outputs/Data Out 12
//     Serial_COM Outputs/GVL_Serial_Com.stComOut_DREAM_DP1_PTM_01/D[13] <-> COM RxPDO-Map Outputs/Data Out 13
//     Serial_COM Outputs/GVL_Serial_Com.stComOut_DREAM_DP1_PTM_01/D[14] <-> COM RxPDO-Map Outputs/Data Out 14
//     Serial_COM Outputs/GVL_Serial_Com.stComOut_DREAM_DP1_PTM_01/D[15] <-> COM RxPDO-Map Outputs/Data Out 15
//     Serial_COM Outputs/GVL_Serial_Com.stComOut_DREAM_DP1_PTM_01/D[16] <-> COM RxPDO-Map Outputs/Data Out 16
//     Serial_COM Outputs/GVL_Serial_Com.stComOut_DREAM_DP1_PTM_01/D[17] <-> COM RxPDO-Map Outputs/Data Out 17
//     Serial_COM Outputs/GVL_Serial_Com.stComOut_DREAM_DP1_PTM_01/D[18] <-> COM RxPDO-Map Outputs/Data Out 18
//     Serial_COM Outputs/GVL_Serial_Com.stComOut_DREAM_DP1_PTM_01/D[19] <-> COM RxPDO-Map Outputs/Data Out 19
//     Serial_COM Outputs/GVL_Serial_Com.stComOut_DREAM_DP1_PTM_01/D[1] <-> COM RxPDO-Map Outputs/Data Out 1
//     Serial_COM Outputs/GVL_Serial_Com.stComOut_DREAM_DP1_PTM_01/D[20] <-> COM RxPDO-Map Outputs/Data Out 20
//     Serial_COM Outputs/GVL_Serial_Com.stComOut_DREAM_DP1_PTM_01/D[21] <-> COM RxPDO-Map Outputs/Data Out 21
//     Serial_COM Outputs/GVL_Serial_Com.stComOut_DREAM_DP1_PTM_01/D[2] <-> COM RxPDO-Map Outputs/Data Out 2
//     Serial_COM Outputs/GVL_Serial_Com.stComOut_DREAM_DP1_PTM_01/D[3] <-> COM RxPDO-Map Outputs/Data Out 3
//     Serial_COM Outputs/GVL_Serial_Com.stComOut_DREAM_DP1_PTM_01/D[4] <-> COM RxPDO-Map Outputs/Data Out 4
//     Serial_COM Outputs/GVL_Serial_Com.stComOut_DREAM_DP1_PTM_01/D[5] <-> COM RxPDO-Map Outputs/Data Out 5
//     Serial_COM Outputs/GVL_Serial_Com.stComOut_DREAM_DP1_PTM_01/D[6] <-> COM RxPDO-Map Outputs/Data Out 6
//     Serial_COM Outputs/GVL_Serial_Com.stComOut_DREAM_DP1_PTM_01/D[7] <-> COM RxPDO-Map Outputs/Data Out 7
//     Serial_COM Outputs/GVL_Serial_Com.stComOut_DREAM_DP1_PTM_01/D[8] <-> COM RxPDO-Map Outputs/Data Out 8
//     Serial_COM Outputs/GVL_Serial_Com.stComOut_DREAM_DP1_PTM_01/D[9] <-> COM RxPDO-Map Outputs/Data Out 9
//   lcls_plc_dream_vac Instance <-> Device 1 (EtherCAT)/R20_DRL_03_CX0_EK1200/R20_DRL_03_E15_EL1122/K4S8_DRL_03_EK0_EK1100/K4S8_DRL_03_E19_EL1004
//     PlcTask Inputs/GVL_VAC_PUMPS.DREAM_DP1_PTM_01.i_xAtSpd <-> Channel 1/Input
//     PlcTask Inputs/GVL_VAC_PUMPS.DREAM_DP1_PTM_01.i_xFaultNC <-> Channel 3/Input
//     PlcTask Inputs/GVL_VAC_PUMPS.DREAM_DP1_PTM_01.i_xRemote <-> Channel 2/Input
//   lcls_plc_dream_vac Instance <-> Device 1 (EtherCAT)/R20_DRL_03_CX0_EK1200/R20_DRL_03_E15_EL1122/K4S8_DRL_03_EK0_EK1100/K4S8_DRL_03_E1_EL2624
//     PlcTask Outputs/GVL_VAC_GAUGES.DREAM_DP1_GHC_01.q_xHV_DIS <-> Channel 2/Output
//     PlcTask Outputs/GVL_VAC_GAUGES.DREAM_DP2_GHC_01.q_xHV_DIS <-> Channel 3/Output
//     PlcTask Outputs/GVL_VAC_GAUGES.DREAM_DP3_GHC_01.q_xHV_DIS <-> Channel 4/Output
//     PlcTask Outputs/GVL_VAC_GAUGES.DREAM_NC_GCC_01.q_xHV_DIS <-> Channel 1/Output
//   lcls_plc_dream_vac Instance <-> Device 1 (EtherCAT)/R20_DRL_03_CX0_EK1200/R20_DRL_03_E15_EL1122/K4S8_DRL_03_EK0_EK1100/K4S8_DRL_03_E20_EL2004
//     PlcTask Outputs/GVL_VAC_PUMPS.DREAM_DP1_PTM_01.q_PumpingStation <-> Channel 3/Output
//     PlcTask Outputs/GVL_VAC_PUMPS.DREAM_DP1_PTM_01.q_RunDO <-> Channel 1/Output
//     PlcTask Outputs/GVL_VAC_PUMPS.DREAM_DP1_PTM_01.q_xRemote <-> Channel 2/Output
//   lcls_plc_dream_vac Instance <-> Device 1 (EtherCAT)/R20_DRL_03_CX0_EK1200/R20_DRL_03_E15_EL1122/K4S8_DRL_03_EK0_EK1100/K4S8_DRL_03_E21_EL3052
//     PlcTask Inputs/GVL_FWM.fbCoilFlowMeter.iRaw <-> AI Standard Channel 1/Value
//   lcls_plc_dream_vac Instance <-> Device 1 (EtherCAT)/R20_DRL_03_CX0_EK1200/R20_DRL_03_E15_EL1122/K4S8_DRL_03_EK0_EK1100/K4S8_DRL_03_E22_EL3314
//     PlcTask Inputs/GVL_TC.TC_01.bError <-> TC Inputs Channel 1/Status/Error
//     PlcTask Inputs/GVL_TC.TC_02.bError <-> TC Inputs Channel 2/Status/Error
//     PlcTask Inputs/GVL_TC.TC_03.bError <-> TC Inputs Channel 3/Status/Error
//     PlcTask Inputs/GVL_TC.TC_04.bError <-> TC Inputs Channel 4/Status/Error
//     PlcTask Inputs/GVL_TC.TC_01.bOverrange <-> TC Inputs Channel 1/Status/Overrange
//     PlcTask Inputs/GVL_TC.TC_02.bOverrange <-> TC Inputs Channel 2/Status/Overrange
//     PlcTask Inputs/GVL_TC.TC_03.bOverrange <-> TC Inputs Channel 3/Status/Overrange
//     PlcTask Inputs/GVL_TC.TC_04.bOverrange <-> TC Inputs Channel 4/Status/Overrange
//     PlcTask Inputs/GVL_TC.TC_01.bUnderrange <-> TC Inputs Channel 1/Status/Underrange
//     PlcTask Inputs/GVL_TC.TC_02.bUnderrange <-> TC Inputs Channel 2/Status/Underrange
//     PlcTask Inputs/GVL_TC.TC_03.bUnderrange <-> TC Inputs Channel 3/Status/Underrange
//     PlcTask Inputs/GVL_TC.TC_04.bUnderrange <-> TC Inputs Channel 4/Status/Underrange
//     PlcTask Inputs/GVL_TC.TC_01.iRaw <-> TC Inputs Channel 1/Value
//     PlcTask Inputs/GVL_TC.TC_02.iRaw <-> TC Inputs Channel 2/Value
//     PlcTask Inputs/GVL_TC.TC_03.iRaw <-> TC Inputs Channel 3/Value
//     PlcTask Inputs/GVL_TC.TC_04.iRaw <-> TC Inputs Channel 4/Value
//   lcls_plc_dream_vac Instance <-> Device 1 (EtherCAT)/R20_DRL_03_CX0_EK1200/R20_DRL_03_E15_EL1122/K4S8_DRL_03_EK0_EK1100/K4S8_DRL_03_E23_EL3314
//     PlcTask Inputs/GVL_TC.TC_05.bError <-> TC Inputs Channel 1/Status/Error
//     PlcTask Inputs/GVL_TC.TC_06.bError <-> TC Inputs Channel 2/Status/Error
//     PlcTask Inputs/GVL_TC.TC_07.bError <-> TC Inputs Channel 3/Status/Error
//     PlcTask Inputs/GVL_TC.TC_08.bError <-> TC Inputs Channel 4/Status/Error
//     PlcTask Inputs/GVL_TC.TC_05.bOverrange <-> TC Inputs Channel 1/Status/Overrange
//     PlcTask Inputs/GVL_TC.TC_06.bOverrange <-> TC Inputs Channel 2/Status/Overrange
//     PlcTask Inputs/GVL_TC.TC_07.bOverrange <-> TC Inputs Channel 3/Status/Overrange
//     PlcTask Inputs/GVL_TC.TC_08.bOverrange <-> TC Inputs Channel 4/Status/Overrange
//     PlcTask Inputs/GVL_TC.TC_05.bUnderrange <-> TC Inputs Channel 1/Status/Underrange
//     PlcTask Inputs/GVL_TC.TC_06.bUnderrange <-> TC Inputs Channel 2/Status/Underrange
//     PlcTask Inputs/GVL_TC.TC_07.bUnderrange <-> TC Inputs Channel 3/Status/Underrange
//     PlcTask Inputs/GVL_TC.TC_08.bUnderrange <-> TC Inputs Channel 4/Status/Underrange
//     PlcTask Inputs/GVL_TC.TC_05.iRaw <-> TC Inputs Channel 1/Value
//     PlcTask Inputs/GVL_TC.TC_06.iRaw <-> TC Inputs Channel 2/Value
//     PlcTask Inputs/GVL_TC.TC_07.iRaw <-> TC Inputs Channel 3/Value
//     PlcTask Inputs/GVL_TC.TC_08.iRaw <-> TC Inputs Channel 4/Value
//   lcls_plc_dream_vac Instance <-> Device 1 (EtherCAT)/R20_DRL_03_CX0_EK1200/R20_DRL_03_E15_EL1122/K4S8_DRL_03_EK0_EK1100/K4S8_DRL_03_E4_EL1084
//     PlcTask Inputs/GVL_VAC_GAUGES.DREAM_DP1_GHC_01.i_xHV_ON <-> Channel 4/Input
//     PlcTask Inputs/GVL_VAC_GAUGES.DREAM_DP2_GHC_01.i_xHV_ON <-> Channel 1/Input
//     PlcTask Inputs/GVL_VAC_GAUGES.DREAM_DP3_GHC_01.i_xHV_ON <-> Channel 2/Input
//     PlcTask Inputs/GVL_VAC_GAUGES.DREAM_NC_GCC_01.i_xHV_ON <-> Channel 3/Input
//   lcls_plc_dream_vac Instance <-> Device 1 (EtherCAT)/R20_DRL_03_CX0_EK1200/R20_DRL_03_E15_EL1122/K4S8_DRL_03_EK0_EK1100/K4S8_DRL_03_E5_EL3174-0002
//     PlcTask Inputs/GVL_VAC_GAUGES.DREAM_DP1_GHC_01.i_iPRESS_R <-> AI Standard Channel 2/Value
//     PlcTask Inputs/GVL_VAC_GAUGES.DREAM_DP2_GHC_01.i_iPRESS_R <-> AI Standard Channel 3/Value
//     PlcTask Inputs/GVL_VAC_GAUGES.DREAM_DP3_GHC_01.i_iPRESS_R <-> AI Standard Channel 4/Value
//     PlcTask Inputs/GVL_VAC_GAUGES.DREAM_NC_GCC_01.i_iPRESS_R <-> AI Standard Channel 1/Value
//   lcls_plc_dream_vac Instance <-> Device 1 (EtherCAT)/R20_DRL_03_CX0_EK1200/R20_DRL_03_E15_EL1122/K4S8_DRL_03_EK0_EK1100/K4S8_DRL_03_E6_EL3174-0002
//     PlcTask Inputs/GVL_VAC_GAUGES.DREAM_DP1_GPI_01.i_iPRESS_R <-> AI Standard Channel 2/Value
//     PlcTask Inputs/GVL_VAC_GAUGES.DREAM_NC_GPI_01.i_iPRESS_R <-> AI Standard Channel 1/Value
//   lcls_plc_dream_vac Instance <-> Device 1 (EtherCAT)/R20_DRL_03_CX0_EK1200/R20_DRL_03_E15_EL1122/K4S8_DRL_04_EK0_EK1100/K4S8_DRL_04_E10_EL1004
//     PlcTask Inputs/GVL_VAC_VALVES.DREAM_ROUGH1_VRC_20.i_xClsLS <-> Channel 4/Input
//     PlcTask Inputs/GVL_VAC_VALVES.DREAM_ROUGH2_VRC_02.i_xClsLS <-> Channel 2/Input
//     PlcTask Inputs/GVL_VAC_VALVES.DREAM_ROUGH1_VRC_20.i_xOpnLS <-> Channel 3/Input
//     PlcTask Inputs/GVL_VAC_VALVES.DREAM_ROUGH2_VRC_02.i_xOpnLS <-> Channel 1/Input
//   lcls_plc_dream_vac Instance <-> Device 1 (EtherCAT)/R20_DRL_03_CX0_EK1200/R20_DRL_03_E15_EL1122/K4S8_DRL_04_EK0_EK1100/K4S8_DRL_04_E11_EL2004
//     PlcTask Outputs/GVL_VAC_VALVES.DREAM_ROUGH1_VRC_01.q_xOPN_DO <-> Channel 1/Output
//     PlcTask Outputs/GVL_VAC_VALVES.DREAM_ROUGH1_VRC_20.q_xOPN_DO <-> Channel 4/Output
//     PlcTask Outputs/GVL_VAC_VALVES.DREAM_ROUGH2_VRC_01.q_xOPN_DO <-> Channel 2/Output
//     PlcTask Outputs/GVL_VAC_VALVES.DREAM_ROUGH2_VRC_02.q_xOPN_DO <-> Channel 3/Output
//   lcls_plc_dream_vac Instance <-> Device 1 (EtherCAT)/R20_DRL_03_CX0_EK1200/R20_DRL_03_E15_EL1122/K4S8_DRL_04_EK0_EK1100/K4S8_DRL_04_E14_EL2624
//     PlcTask Outputs/GVL_PLC_Interface.bCoilPS_ILK <-> Channel 3/Output
//     PlcTask Outputs/GVL_PLC_Interface.bHVSafteyLoopEnable <-> Channel 4/Output
//     PlcTask Outputs/GVL_VAC_GAUGES.DREAM_CAT1_GHC_01.q_xHV_DIS <-> Channel 1/Output
//     PlcTask Outputs/GVL_VAC_GAUGES.DREAM_CAT2_GHC_01.q_xHV_DIS <-> Channel 2/Output
//   lcls_plc_dream_vac Instance <-> Device 1 (EtherCAT)/R20_DRL_03_CX0_EK1200/R20_DRL_03_E15_EL1122/K4S8_DRL_04_EK0_EK1100/K4S8_DRL_04_E15_EL1084
//     PlcTask Inputs/GVL_VAC_GAUGES.DREAM_CAT1_GHC_01.i_xHV_ON <-> Channel 1/Input
//     PlcTask Inputs/GVL_VAC_GAUGES.DREAM_CAT2_GHC_01.i_xHV_ON <-> Channel 2/Input
//   lcls_plc_dream_vac Instance <-> Device 1 (EtherCAT)/R20_DRL_03_CX0_EK1200/R20_DRL_03_E15_EL1122/K4S8_DRL_04_EK0_EK1100/K4S8_DRL_04_E16_EL3174-0002
//     PlcTask Inputs/GVL_FWM.fbCoilCurrentMonitoring.iRaw <-> AI Standard Channel 4/Value
//     PlcTask Inputs/GVL_VAC_GAUGES.DREAM_CAT1_GHC_01.i_iPRESS_R <-> AI Standard Channel 2/Value
//     PlcTask Inputs/GVL_VAC_GAUGES.DREAM_CAT2_GHC_01.i_iPRESS_R <-> AI Standard Channel 3/Value
//     PlcTask Inputs/GVL_VAC_GAUGES.DREAM_MC_GPI_01.i_iPRESS_R <-> AI Standard Channel 1/Value
//   lcls_plc_dream_vac Instance <-> Device 1 (EtherCAT)/R20_DRL_03_CX0_EK1200/R20_DRL_03_E15_EL1122/K4S8_DRL_04_EK0_EK1100/K4S8_DRL_04_E17_EL6001
//     Serial_COM Inputs/GVL_Serial_Com.stComIn_DREAM_ROUGH2_PTM_02/D[0] <-> COM Inputs/Data In 0
//     Serial_COM Inputs/GVL_Serial_Com.stComIn_DREAM_ROUGH2_PTM_02/D[10] <-> COM Inputs/Data In 10
//     Serial_COM Inputs/GVL_Serial_Com.stComIn_DREAM_ROUGH2_PTM_02/D[11] <-> COM Inputs/Data In 11
//     Serial_COM Inputs/GVL_Serial_Com.stComIn_DREAM_ROUGH2_PTM_02/D[12] <-> COM Inputs/Data In 12
//     Serial_COM Inputs/GVL_Serial_Com.stComIn_DREAM_ROUGH2_PTM_02/D[13] <-> COM Inputs/Data In 13
//     Serial_COM Inputs/GVL_Serial_Com.stComIn_DREAM_ROUGH2_PTM_02/D[14] <-> COM Inputs/Data In 14
//     Serial_COM Inputs/GVL_Serial_Com.stComIn_DREAM_ROUGH2_PTM_02/D[15] <-> COM Inputs/Data In 15
//     Serial_COM Inputs/GVL_Serial_Com.stComIn_DREAM_ROUGH2_PTM_02/D[16] <-> COM Inputs/Data In 16
//     Serial_COM Inputs/GVL_Serial_Com.stComIn_DREAM_ROUGH2_PTM_02/D[17] <-> COM Inputs/Data In 17
//     Serial_COM Inputs/GVL_Serial_Com.stComIn_DREAM_ROUGH2_PTM_02/D[18] <-> COM Inputs/Data In 18
//     Serial_COM Inputs/GVL_Serial_Com.stComIn_DREAM_ROUGH2_PTM_02/D[19] <-> COM Inputs/Data In 19
//     Serial_COM Inputs/GVL_Serial_Com.stComIn_DREAM_ROUGH2_PTM_02/D[1] <-> COM Inputs/Data In 1
//     Serial_COM Inputs/GVL_Serial_Com.stComIn_DREAM_ROUGH2_PTM_02/D[20] <-> COM Inputs/Data In 20
//     Serial_COM Inputs/GVL_Serial_Com.stComIn_DREAM_ROUGH2_PTM_02/D[21] <-> COM Inputs/Data In 21
//     Serial_COM Inputs/GVL_Serial_Com.stComIn_DREAM_ROUGH2_PTM_02/D[2] <-> COM Inputs/Data In 2
//     Serial_COM Inputs/GVL_Serial_Com.stComIn_DREAM_ROUGH2_PTM_02/D[3] <-> COM Inputs/Data In 3
//     Serial_COM Inputs/GVL_Serial_Com.stComIn_DREAM_ROUGH2_PTM_02/D[4] <-> COM Inputs/Data In 4
//     Serial_COM Inputs/GVL_Serial_Com.stComIn_DREAM_ROUGH2_PTM_02/D[5] <-> COM Inputs/Data In 5
//     Serial_COM Inputs/GVL_Serial_Com.stComIn_DREAM_ROUGH2_PTM_02/D[6] <-> COM Inputs/Data In 6
//     Serial_COM Inputs/GVL_Serial_Com.stComIn_DREAM_ROUGH2_PTM_02/D[7] <-> COM Inputs/Data In 7
//     Serial_COM Inputs/GVL_Serial_Com.stComIn_DREAM_ROUGH2_PTM_02/D[8] <-> COM Inputs/Data In 8
//     Serial_COM Inputs/GVL_Serial_Com.stComIn_DREAM_ROUGH2_PTM_02/D[9] <-> COM Inputs/Data In 9
//     Serial_COM Inputs/GVL_Serial_Com.stComIn_DREAM_ROUGH2_PTM_02/Status <-> COM Inputs/Status
//     Serial_COM Outputs/GVL_Serial_Com.stComOut_DREAM_ROUGH2_PTM_02/Ctrl <-> COM Outputs/Ctrl
//     Serial_COM Outputs/GVL_Serial_Com.stComOut_DREAM_ROUGH2_PTM_02/D[0] <-> COM Outputs/Data Out 0
//     Serial_COM Outputs/GVL_Serial_Com.stComOut_DREAM_ROUGH2_PTM_02/D[10] <-> COM Outputs/Data Out 10
//     Serial_COM Outputs/GVL_Serial_Com.stComOut_DREAM_ROUGH2_PTM_02/D[11] <-> COM Outputs/Data Out 11
//     Serial_COM Outputs/GVL_Serial_Com.stComOut_DREAM_ROUGH2_PTM_02/D[12] <-> COM Outputs/Data Out 12
//     Serial_COM Outputs/GVL_Serial_Com.stComOut_DREAM_ROUGH2_PTM_02/D[13] <-> COM Outputs/Data Out 13
//     Serial_COM Outputs/GVL_Serial_Com.stComOut_DREAM_ROUGH2_PTM_02/D[14] <-> COM Outputs/Data Out 14
//     Serial_COM Outputs/GVL_Serial_Com.stComOut_DREAM_ROUGH2_PTM_02/D[15] <-> COM Outputs/Data Out 15
//     Serial_COM Outputs/GVL_Serial_Com.stComOut_DREAM_ROUGH2_PTM_02/D[16] <-> COM Outputs/Data Out 16
//     Serial_COM Outputs/GVL_Serial_Com.stComOut_DREAM_ROUGH2_PTM_02/D[17] <-> COM Outputs/Data Out 17
//     Serial_COM Outputs/GVL_Serial_Com.stComOut_DREAM_ROUGH2_PTM_02/D[18] <-> COM Outputs/Data Out 18
//     Serial_COM Outputs/GVL_Serial_Com.stComOut_DREAM_ROUGH2_PTM_02/D[19] <-> COM Outputs/Data Out 19
//     Serial_COM Outputs/GVL_Serial_Com.stComOut_DREAM_ROUGH2_PTM_02/D[1] <-> COM Outputs/Data Out 1
//     Serial_COM Outputs/GVL_Serial_Com.stComOut_DREAM_ROUGH2_PTM_02/D[20] <-> COM Outputs/Data Out 20
//     Serial_COM Outputs/GVL_Serial_Com.stComOut_DREAM_ROUGH2_PTM_02/D[21] <-> COM Outputs/Data Out 21
//     Serial_COM Outputs/GVL_Serial_Com.stComOut_DREAM_ROUGH2_PTM_02/D[2] <-> COM Outputs/Data Out 2
//     Serial_COM Outputs/GVL_Serial_Com.stComOut_DREAM_ROUGH2_PTM_02/D[3] <-> COM Outputs/Data Out 3
//     Serial_COM Outputs/GVL_Serial_Com.stComOut_DREAM_ROUGH2_PTM_02/D[4] <-> COM Outputs/Data Out 4
//     Serial_COM Outputs/GVL_Serial_Com.stComOut_DREAM_ROUGH2_PTM_02/D[5] <-> COM Outputs/Data Out 5
//     Serial_COM Outputs/GVL_Serial_Com.stComOut_DREAM_ROUGH2_PTM_02/D[6] <-> COM Outputs/Data Out 6
//     Serial_COM Outputs/GVL_Serial_Com.stComOut_DREAM_ROUGH2_PTM_02/D[7] <-> COM Outputs/Data Out 7
//     Serial_COM Outputs/GVL_Serial_Com.stComOut_DREAM_ROUGH2_PTM_02/D[8] <-> COM Outputs/Data Out 8
//     Serial_COM Outputs/GVL_Serial_Com.stComOut_DREAM_ROUGH2_PTM_02/D[9] <-> COM Outputs/Data Out 9
//   lcls_plc_dream_vac Instance <-> Device 1 (EtherCAT)/R20_DRL_03_CX0_EK1200/R20_DRL_03_E15_EL1122/K4S8_DRL_04_EK0_EK1100/K4S8_DRL_04_E1_EL1004
//     PlcTask Inputs/GVL_VAC_VALVES.DREAM_CAT1_VRC_01.i_xClsLS <-> Channel 2/Input
//     PlcTask Inputs/GVL_VAC_VALVES.DREAM_CAT1_VRC_01.i_xOpnLS <-> Channel 1/Input
//     PlcTask Inputs/GVL_VAC_VALVES.DREAM_DP1_VRC_20.i_xClsLS <-> Channel 4/Input
//     PlcTask Inputs/GVL_VAC_VALVES.DREAM_DP1_VRC_20.i_xOpnLS <-> Channel 3/Input
//   lcls_plc_dream_vac Instance <-> Device 1 (EtherCAT)/R20_DRL_03_CX0_EK1200/R20_DRL_03_E15_EL1122/K4S8_DRL_04_EK0_EK1100/K4S8_DRL_04_E2_EL2004
//     PlcTask Outputs/GVL_VAC_VALVES.DREAM_CAT1_VRC_01.q_xOPN_DO <-> Channel 1/Output
//     PlcTask Outputs/GVL_VAC_VALVES.DREAM_DP1_VRC_20.q_xCLS_DO <-> Channel 4/Output
//     PlcTask Outputs/GVL_VAC_VALVES.DREAM_DP1_VRC_20.q_xOPN_DO <-> Channel 3/Output
//   lcls_plc_dream_vac Instance <-> Device 1 (EtherCAT)/R20_DRL_03_CX0_EK1200/R20_DRL_03_E15_EL1122/K4S8_DRL_04_EK0_EK1100/K4S8_DRL_04_E3_EL1004
//     PlcTask Inputs/GVL_VAC_PUMPS.DREAM_CAT1_PTM_01.i_xAtSpd <-> Channel 4/Input
//     PlcTask Inputs/GVL_VAC_PUMPS.DREAM_CAT1_PTM_01.i_xFaultNC <-> Channel 3/Input
//     PlcTask Inputs/GVL_VAC_PUMPS.DREAM_ROUGH2_PTM_01.i_xAtSpd <-> Channel 2/Input
//     PlcTask Inputs/GVL_VAC_PUMPS.DREAM_ROUGH2_PTM_01.i_xFaultNC <-> Channel 1/Input
//   lcls_plc_dream_vac Instance <-> Device 1 (EtherCAT)/R20_DRL_03_CX0_EK1200/R20_DRL_03_E15_EL1122/K4S8_DRL_04_EK0_EK1100/K4S8_DRL_04_E4_EL1004
//     PlcTask Inputs/GVL_VAC_PUMPS.DREAM_CAT2_PTM_01.i_xAtSpd <-> Channel 2/Input
//     PlcTask Inputs/GVL_VAC_PUMPS.DREAM_CAT2_PTM_01.i_xFaultNC <-> Channel 1/Input
//     PlcTask Inputs/GVL_VAC_PUMPS.DREAM_ROUGH2_PTM_02.i_xAtSpd <-> Channel 4/Input
//     PlcTask Inputs/GVL_VAC_PUMPS.DREAM_ROUGH2_PTM_02.i_xFaultNC <-> Channel 3/Input
//   lcls_plc_dream_vac Instance <-> Device 1 (EtherCAT)/R20_DRL_03_CX0_EK1200/R20_DRL_03_E15_EL1122/K4S8_DRL_04_EK0_EK1100/K4S8_DRL_04_E5_EL2794
//     PlcTask Outputs/GVL_VAC_PUMPS.DREAM_CAT1_PTM_01.q_RunDO <-> Channel 2/Output
//     PlcTask Outputs/GVL_VAC_PUMPS.DREAM_CAT2_PTM_01.q_RunDO <-> Channel 3/Output
//     PlcTask Outputs/GVL_VAC_PUMPS.DREAM_ROUGH2_PTM_01.q_RunDO <-> Channel 1/Output
//     PlcTask Outputs/GVL_VAC_PUMPS.DREAM_ROUGH2_PTM_02.q_RunDO <-> Channel 4/Output
//   lcls_plc_dream_vac Instance <-> Device 1 (EtherCAT)/R20_DRL_03_CX0_EK1200/R20_DRL_03_E15_EL1122/K4S8_DRL_04_EK0_EK1100/K4S8_DRL_04_E6_EL6001
//     Serial_COM Inputs/GVL_Serial_Com.stComIn_DREAM_ROUGH2_PTM_01/D[0] <-> COM Inputs/Data In 0
//     Serial_COM Inputs/GVL_Serial_Com.stComIn_DREAM_ROUGH2_PTM_01/D[10] <-> COM Inputs/Data In 10
//     Serial_COM Inputs/GVL_Serial_Com.stComIn_DREAM_ROUGH2_PTM_01/D[11] <-> COM Inputs/Data In 11
//     Serial_COM Inputs/GVL_Serial_Com.stComIn_DREAM_ROUGH2_PTM_01/D[12] <-> COM Inputs/Data In 12
//     Serial_COM Inputs/GVL_Serial_Com.stComIn_DREAM_ROUGH2_PTM_01/D[13] <-> COM Inputs/Data In 13
//     Serial_COM Inputs/GVL_Serial_Com.stComIn_DREAM_ROUGH2_PTM_01/D[14] <-> COM Inputs/Data In 14
//     Serial_COM Inputs/GVL_Serial_Com.stComIn_DREAM_ROUGH2_PTM_01/D[15] <-> COM Inputs/Data In 15
//     Serial_COM Inputs/GVL_Serial_Com.stComIn_DREAM_ROUGH2_PTM_01/D[16] <-> COM Inputs/Data In 16
//     Serial_COM Inputs/GVL_Serial_Com.stComIn_DREAM_ROUGH2_PTM_01/D[17] <-> COM Inputs/Data In 17
//     Serial_COM Inputs/GVL_Serial_Com.stComIn_DREAM_ROUGH2_PTM_01/D[18] <-> COM Inputs/Data In 18
//     Serial_COM Inputs/GVL_Serial_Com.stComIn_DREAM_ROUGH2_PTM_01/D[19] <-> COM Inputs/Data In 19
//     Serial_COM Inputs/GVL_Serial_Com.stComIn_DREAM_ROUGH2_PTM_01/D[1] <-> COM Inputs/Data In 1
//     Serial_COM Inputs/GVL_Serial_Com.stComIn_DREAM_ROUGH2_PTM_01/D[20] <-> COM Inputs/Data In 20
//     Serial_COM Inputs/GVL_Serial_Com.stComIn_DREAM_ROUGH2_PTM_01/D[21] <-> COM Inputs/Data In 21
//     Serial_COM Inputs/GVL_Serial_Com.stComIn_DREAM_ROUGH2_PTM_01/D[2] <-> COM Inputs/Data In 2
//     Serial_COM Inputs/GVL_Serial_Com.stComIn_DREAM_ROUGH2_PTM_01/D[3] <-> COM Inputs/Data In 3
//     Serial_COM Inputs/GVL_Serial_Com.stComIn_DREAM_ROUGH2_PTM_01/D[4] <-> COM Inputs/Data In 4
//     Serial_COM Inputs/GVL_Serial_Com.stComIn_DREAM_ROUGH2_PTM_01/D[5] <-> COM Inputs/Data In 5
//     Serial_COM Inputs/GVL_Serial_Com.stComIn_DREAM_ROUGH2_PTM_01/D[6] <-> COM Inputs/Data In 6
//     Serial_COM Inputs/GVL_Serial_Com.stComIn_DREAM_ROUGH2_PTM_01/D[7] <-> COM Inputs/Data In 7
//     Serial_COM Inputs/GVL_Serial_Com.stComIn_DREAM_ROUGH2_PTM_01/D[8] <-> COM Inputs/Data In 8
//     Serial_COM Inputs/GVL_Serial_Com.stComIn_DREAM_ROUGH2_PTM_01/D[9] <-> COM Inputs/Data In 9
//     Serial_COM Inputs/GVL_Serial_Com.stComIn_DREAM_ROUGH2_PTM_01/Status <-> COM Inputs/Status
//     Serial_COM Outputs/GVL_Serial_Com.stComOut_DREAM_ROUGH2_PTM_01/Ctrl <-> COM Outputs/Ctrl
//     Serial_COM Outputs/GVL_Serial_Com.stComOut_DREAM_ROUGH2_PTM_01/D[0] <-> COM Outputs/Data Out 0
//     Serial_COM Outputs/GVL_Serial_Com.stComOut_DREAM_ROUGH2_PTM_01/D[10] <-> COM Outputs/Data Out 10
//     Serial_COM Outputs/GVL_Serial_Com.stComOut_DREAM_ROUGH2_PTM_01/D[11] <-> COM Outputs/Data Out 11
//     Serial_COM Outputs/GVL_Serial_Com.stComOut_DREAM_ROUGH2_PTM_01/D[12] <-> COM Outputs/Data Out 12
//     Serial_COM Outputs/GVL_Serial_Com.stComOut_DREAM_ROUGH2_PTM_01/D[13] <-> COM Outputs/Data Out 13
//     Serial_COM Outputs/GVL_Serial_Com.stComOut_DREAM_ROUGH2_PTM_01/D[14] <-> COM Outputs/Data Out 14
//     Serial_COM Outputs/GVL_Serial_Com.stComOut_DREAM_ROUGH2_PTM_01/D[15] <-> COM Outputs/Data Out 15
//     Serial_COM Outputs/GVL_Serial_Com.stComOut_DREAM_ROUGH2_PTM_01/D[16] <-> COM Outputs/Data Out 16
//     Serial_COM Outputs/GVL_Serial_Com.stComOut_DREAM_ROUGH2_PTM_01/D[17] <-> COM Outputs/Data Out 17
//     Serial_COM Outputs/GVL_Serial_Com.stComOut_DREAM_ROUGH2_PTM_01/D[18] <-> COM Outputs/Data Out 18
//     Serial_COM Outputs/GVL_Serial_Com.stComOut_DREAM_ROUGH2_PTM_01/D[19] <-> COM Outputs/Data Out 19
//     Serial_COM Outputs/GVL_Serial_Com.stComOut_DREAM_ROUGH2_PTM_01/D[1] <-> COM Outputs/Data Out 1
//     Serial_COM Outputs/GVL_Serial_Com.stComOut_DREAM_ROUGH2_PTM_01/D[20] <-> COM Outputs/Data Out 20
//     Serial_COM Outputs/GVL_Serial_Com.stComOut_DREAM_ROUGH2_PTM_01/D[21] <-> COM Outputs/Data Out 21
//     Serial_COM Outputs/GVL_Serial_Com.stComOut_DREAM_ROUGH2_PTM_01/D[2] <-> COM Outputs/Data Out 2
//     Serial_COM Outputs/GVL_Serial_Com.stComOut_DREAM_ROUGH2_PTM_01/D[3] <-> COM Outputs/Data Out 3
//     Serial_COM Outputs/GVL_Serial_Com.stComOut_DREAM_ROUGH2_PTM_01/D[4] <-> COM Outputs/Data Out 4
//     Serial_COM Outputs/GVL_Serial_Com.stComOut_DREAM_ROUGH2_PTM_01/D[5] <-> COM Outputs/Data Out 5
//     Serial_COM Outputs/GVL_Serial_Com.stComOut_DREAM_ROUGH2_PTM_01/D[6] <-> COM Outputs/Data Out 6
//     Serial_COM Outputs/GVL_Serial_Com.stComOut_DREAM_ROUGH2_PTM_01/D[7] <-> COM Outputs/Data Out 7
//     Serial_COM Outputs/GVL_Serial_Com.stComOut_DREAM_ROUGH2_PTM_01/D[8] <-> COM Outputs/Data Out 8
//     Serial_COM Outputs/GVL_Serial_Com.stComOut_DREAM_ROUGH2_PTM_01/D[9] <-> COM Outputs/Data Out 9
//   lcls_plc_dream_vac Instance <-> Device 1 (EtherCAT)/R20_DRL_03_CX0_EK1200/R20_DRL_03_E15_EL1122/K4S8_DRL_04_EK0_EK1100/K4S8_DRL_04_E7_EL6001
//     Serial_COM Inputs/GVL_Serial_Com.stComIn_DREAM_CAT1_PTM_01/D[0] <-> COM Inputs/Data In 0
//     Serial_COM Inputs/GVL_Serial_Com.stComIn_DREAM_CAT1_PTM_01/D[10] <-> COM Inputs/Data In 10
//     Serial_COM Inputs/GVL_Serial_Com.stComIn_DREAM_CAT1_PTM_01/D[11] <-> COM Inputs/Data In 11
//     Serial_COM Inputs/GVL_Serial_Com.stComIn_DREAM_CAT1_PTM_01/D[12] <-> COM Inputs/Data In 12
//     Serial_COM Inputs/GVL_Serial_Com.stComIn_DREAM_CAT1_PTM_01/D[13] <-> COM Inputs/Data In 13
//     Serial_COM Inputs/GVL_Serial_Com.stComIn_DREAM_CAT1_PTM_01/D[14] <-> COM Inputs/Data In 14
//     Serial_COM Inputs/GVL_Serial_Com.stComIn_DREAM_CAT1_PTM_01/D[15] <-> COM Inputs/Data In 15
//     Serial_COM Inputs/GVL_Serial_Com.stComIn_DREAM_CAT1_PTM_01/D[16] <-> COM Inputs/Data In 16
//     Serial_COM Inputs/GVL_Serial_Com.stComIn_DREAM_CAT1_PTM_01/D[17] <-> COM Inputs/Data In 17
//     Serial_COM Inputs/GVL_Serial_Com.stComIn_DREAM_CAT1_PTM_01/D[18] <-> COM Inputs/Data In 18
//     Serial_COM Inputs/GVL_Serial_Com.stComIn_DREAM_CAT1_PTM_01/D[19] <-> COM Inputs/Data In 19
//     Serial_COM Inputs/GVL_Serial_Com.stComIn_DREAM_CAT1_PTM_01/D[1] <-> COM Inputs/Data In 1
//     Serial_COM Inputs/GVL_Serial_Com.stComIn_DREAM_CAT1_PTM_01/D[20] <-> COM Inputs/Data In 20
//     Serial_COM Inputs/GVL_Serial_Com.stComIn_DREAM_CAT1_PTM_01/D[21] <-> COM Inputs/Data In 21
//     Serial_COM Inputs/GVL_Serial_Com.stComIn_DREAM_CAT1_PTM_01/D[2] <-> COM Inputs/Data In 2
//     Serial_COM Inputs/GVL_Serial_Com.stComIn_DREAM_CAT1_PTM_01/D[3] <-> COM Inputs/Data In 3
//     Serial_COM Inputs/GVL_Serial_Com.stComIn_DREAM_CAT1_PTM_01/D[4] <-> COM Inputs/Data In 4
//     Serial_COM Inputs/GVL_Serial_Com.stComIn_DREAM_CAT1_PTM_01/D[5] <-> COM Inputs/Data In 5
//     Serial_COM Inputs/GVL_Serial_Com.stComIn_DREAM_CAT1_PTM_01/D[6] <-> COM Inputs/Data In 6
//     Serial_COM Inputs/GVL_Serial_Com.stComIn_DREAM_CAT1_PTM_01/D[7] <-> COM Inputs/Data In 7
//     Serial_COM Inputs/GVL_Serial_Com.stComIn_DREAM_CAT1_PTM_01/D[8] <-> COM Inputs/Data In 8
//     Serial_COM Inputs/GVL_Serial_Com.stComIn_DREAM_CAT1_PTM_01/D[9] <-> COM Inputs/Data In 9
//     Serial_COM Inputs/GVL_Serial_Com.stComIn_DREAM_CAT1_PTM_01/Status <-> COM Inputs/Status
//     Serial_COM Outputs/GVL_Serial_Com.stComOut_DREAM_CAT1_PTM_01/Ctrl <-> COM Outputs/Ctrl
//     Serial_COM Outputs/GVL_Serial_Com.stComOut_DREAM_CAT1_PTM_01/D[0] <-> COM Outputs/Data Out 0
//     Serial_COM Outputs/GVL_Serial_Com.stComOut_DREAM_CAT1_PTM_01/D[10] <-> COM Outputs/Data Out 10
//     Serial_COM Outputs/GVL_Serial_Com.stComOut_DREAM_CAT1_PTM_01/D[11] <-> COM Outputs/Data Out 11
//     Serial_COM Outputs/GVL_Serial_Com.stComOut_DREAM_CAT1_PTM_01/D[12] <-> COM Outputs/Data Out 12
//     Serial_COM Outputs/GVL_Serial_Com.stComOut_DREAM_CAT1_PTM_01/D[13] <-> COM Outputs/Data Out 13
//     Serial_COM Outputs/GVL_Serial_Com.stComOut_DREAM_CAT1_PTM_01/D[14] <-> COM Outputs/Data Out 14
//     Serial_COM Outputs/GVL_Serial_Com.stComOut_DREAM_CAT1_PTM_01/D[15] <-> COM Outputs/Data Out 15
//     Serial_COM Outputs/GVL_Serial_Com.stComOut_DREAM_CAT1_PTM_01/D[16] <-> COM Outputs/Data Out 16
//     Serial_COM Outputs/GVL_Serial_Com.stComOut_DREAM_CAT1_PTM_01/D[17] <-> COM Outputs/Data Out 17
//     Serial_COM Outputs/GVL_Serial_Com.stComOut_DREAM_CAT1_PTM_01/D[18] <-> COM Outputs/Data Out 18
//     Serial_COM Outputs/GVL_Serial_Com.stComOut_DREAM_CAT1_PTM_01/D[19] <-> COM Outputs/Data Out 19
//     Serial_COM Outputs/GVL_Serial_Com.stComOut_DREAM_CAT1_PTM_01/D[1] <-> COM Outputs/Data Out 1
//     Serial_COM Outputs/GVL_Serial_Com.stComOut_DREAM_CAT1_PTM_01/D[20] <-> COM Outputs/Data Out 20
//     Serial_COM Outputs/GVL_Serial_Com.stComOut_DREAM_CAT1_PTM_01/D[21] <-> COM Outputs/Data Out 21
//     Serial_COM Outputs/GVL_Serial_Com.stComOut_DREAM_CAT1_PTM_01/D[2] <-> COM Outputs/Data Out 2
//     Serial_COM Outputs/GVL_Serial_Com.stComOut_DREAM_CAT1_PTM_01/D[3] <-> COM Outputs/Data Out 3
//     Serial_COM Outputs/GVL_Serial_Com.stComOut_DREAM_CAT1_PTM_01/D[4] <-> COM Outputs/Data Out 4
//     Serial_COM Outputs/GVL_Serial_Com.stComOut_DREAM_CAT1_PTM_01/D[5] <-> COM Outputs/Data Out 5
//     Serial_COM Outputs/GVL_Serial_Com.stComOut_DREAM_CAT1_PTM_01/D[6] <-> COM Outputs/Data Out 6
//     Serial_COM Outputs/GVL_Serial_Com.stComOut_DREAM_CAT1_PTM_01/D[7] <-> COM Outputs/Data Out 7
//     Serial_COM Outputs/GVL_Serial_Com.stComOut_DREAM_CAT1_PTM_01/D[8] <-> COM Outputs/Data Out 8
//     Serial_COM Outputs/GVL_Serial_Com.stComOut_DREAM_CAT1_PTM_01/D[9] <-> COM Outputs/Data Out 9
//   lcls_plc_dream_vac Instance <-> Device 1 (EtherCAT)/R20_DRL_03_CX0_EK1200/R20_DRL_03_E15_EL1122/K4S8_DRL_04_EK0_EK1100/K4S8_DRL_04_E8_EL6001
//     Serial_COM Inputs/GVL_Serial_Com.stComIn_DREAM_CAT2_PTM_01/D[0] <-> COM Inputs/Data In 0
//     Serial_COM Inputs/GVL_Serial_Com.stComIn_DREAM_CAT2_PTM_01/D[10] <-> COM Inputs/Data In 10
//     Serial_COM Inputs/GVL_Serial_Com.stComIn_DREAM_CAT2_PTM_01/D[11] <-> COM Inputs/Data In 11
//     Serial_COM Inputs/GVL_Serial_Com.stComIn_DREAM_CAT2_PTM_01/D[12] <-> COM Inputs/Data In 12
//     Serial_COM Inputs/GVL_Serial_Com.stComIn_DREAM_CAT2_PTM_01/D[13] <-> COM Inputs/Data In 13
//     Serial_COM Inputs/GVL_Serial_Com.stComIn_DREAM_CAT2_PTM_01/D[14] <-> COM Inputs/Data In 14
//     Serial_COM Inputs/GVL_Serial_Com.stComIn_DREAM_CAT2_PTM_01/D[15] <-> COM Inputs/Data In 15
//     Serial_COM Inputs/GVL_Serial_Com.stComIn_DREAM_CAT2_PTM_01/D[16] <-> COM Inputs/Data In 16
//     Serial_COM Inputs/GVL_Serial_Com.stComIn_DREAM_CAT2_PTM_01/D[17] <-> COM Inputs/Data In 17
//     Serial_COM Inputs/GVL_Serial_Com.stComIn_DREAM_CAT2_PTM_01/D[18] <-> COM Inputs/Data In 18
//     Serial_COM Inputs/GVL_Serial_Com.stComIn_DREAM_CAT2_PTM_01/D[19] <-> COM Inputs/Data In 19
//     Serial_COM Inputs/GVL_Serial_Com.stComIn_DREAM_CAT2_PTM_01/D[1] <-> COM Inputs/Data In 1
//     Serial_COM Inputs/GVL_Serial_Com.stComIn_DREAM_CAT2_PTM_01/D[20] <-> COM Inputs/Data In 20
//     Serial_COM Inputs/GVL_Serial_Com.stComIn_DREAM_CAT2_PTM_01/D[21] <-> COM Inputs/Data In 21
//     Serial_COM Inputs/GVL_Serial_Com.stComIn_DREAM_CAT2_PTM_01/D[2] <-> COM Inputs/Data In 2
//     Serial_COM Inputs/GVL_Serial_Com.stComIn_DREAM_CAT2_PTM_01/D[3] <-> COM Inputs/Data In 3
//     Serial_COM Inputs/GVL_Serial_Com.stComIn_DREAM_CAT2_PTM_01/D[4] <-> COM Inputs/Data In 4
//     Serial_COM Inputs/GVL_Serial_Com.stComIn_DREAM_CAT2_PTM_01/D[5] <-> COM Inputs/Data In 5
//     Serial_COM Inputs/GVL_Serial_Com.stComIn_DREAM_CAT2_PTM_01/D[6] <-> COM Inputs/Data In 6
//     Serial_COM Inputs/GVL_Serial_Com.stComIn_DREAM_CAT2_PTM_01/D[7] <-> COM Inputs/Data In 7
//     Serial_COM Inputs/GVL_Serial_Com.stComIn_DREAM_CAT2_PTM_01/D[8] <-> COM Inputs/Data In 8
//     Serial_COM Inputs/GVL_Serial_Com.stComIn_DREAM_CAT2_PTM_01/D[9] <-> COM Inputs/Data In 9
//     Serial_COM Inputs/GVL_Serial_Com.stComIn_DREAM_CAT2_PTM_01/Status <-> COM Inputs/Status
//     Serial_COM Outputs/GVL_Serial_Com.stComOut_DREAM_CAT2_PTM_01/Ctrl <-> COM Outputs/Ctrl
//     Serial_COM Outputs/GVL_Serial_Com.stComOut_DREAM_CAT2_PTM_01/D[0] <-> COM Outputs/Data Out 0
//     Serial_COM Outputs/GVL_Serial_Com.stComOut_DREAM_CAT2_PTM_01/D[10] <-> COM Outputs/Data Out 10
//     Serial_COM Outputs/GVL_Serial_Com.stComOut_DREAM_CAT2_PTM_01/D[11] <-> COM Outputs/Data Out 11
//     Serial_COM Outputs/GVL_Serial_Com.stComOut_DREAM_CAT2_PTM_01/D[12] <-> COM Outputs/Data Out 12
//     Serial_COM Outputs/GVL_Serial_Com.stComOut_DREAM_CAT2_PTM_01/D[13] <-> COM Outputs/Data Out 13
//     Serial_COM Outputs/GVL_Serial_Com.stComOut_DREAM_CAT2_PTM_01/D[14] <-> COM Outputs/Data Out 14
//     Serial_COM Outputs/GVL_Serial_Com.stComOut_DREAM_CAT2_PTM_01/D[15] <-> COM Outputs/Data Out 15
//     Serial_COM Outputs/GVL_Serial_Com.stComOut_DREAM_CAT2_PTM_01/D[16] <-> COM Outputs/Data Out 16
//     Serial_COM Outputs/GVL_Serial_Com.stComOut_DREAM_CAT2_PTM_01/D[17] <-> COM Outputs/Data Out 17
//     Serial_COM Outputs/GVL_Serial_Com.stComOut_DREAM_CAT2_PTM_01/D[18] <-> COM Outputs/Data Out 18
//     Serial_COM Outputs/GVL_Serial_Com.stComOut_DREAM_CAT2_PTM_01/D[19] <-> COM Outputs/Data Out 19
//     Serial_COM Outputs/GVL_Serial_Com.stComOut_DREAM_CAT2_PTM_01/D[1] <-> COM Outputs/Data Out 1
//     Serial_COM Outputs/GVL_Serial_Com.stComOut_DREAM_CAT2_PTM_01/D[20] <-> COM Outputs/Data Out 20
//     Serial_COM Outputs/GVL_Serial_Com.stComOut_DREAM_CAT2_PTM_01/D[21] <-> COM Outputs/Data Out 21
//     Serial_COM Outputs/GVL_Serial_Com.stComOut_DREAM_CAT2_PTM_01/D[2] <-> COM Outputs/Data Out 2
//     Serial_COM Outputs/GVL_Serial_Com.stComOut_DREAM_CAT2_PTM_01/D[3] <-> COM Outputs/Data Out 3
//     Serial_COM Outputs/GVL_Serial_Com.stComOut_DREAM_CAT2_PTM_01/D[4] <-> COM Outputs/Data Out 4
//     Serial_COM Outputs/GVL_Serial_Com.stComOut_DREAM_CAT2_PTM_01/D[5] <-> COM Outputs/Data Out 5
//     Serial_COM Outputs/GVL_Serial_Com.stComOut_DREAM_CAT2_PTM_01/D[6] <-> COM Outputs/Data Out 6
//     Serial_COM Outputs/GVL_Serial_Com.stComOut_DREAM_CAT2_PTM_01/D[7] <-> COM Outputs/Data Out 7
//     Serial_COM Outputs/GVL_Serial_Com.stComOut_DREAM_CAT2_PTM_01/D[8] <-> COM Outputs/Data Out 8
//     Serial_COM Outputs/GVL_Serial_Com.stComOut_DREAM_CAT2_PTM_01/D[9] <-> COM Outputs/Data Out 9
//   lcls_plc_dream_vac Instance <-> Device 1 (EtherCAT)/R20_DRL_03_CX0_EK1200/R20_DRL_03_E15_EL1122/K4S8_DRL_04_EK0_EK1100/K4S8_DRL_04_E9_EL1004
//     PlcTask Inputs/GVL_VAC_VALVES.DREAM_ROUGH1_VRC_01.i_xClsLS <-> Channel 2/Input
//     PlcTask Inputs/GVL_VAC_VALVES.DREAM_ROUGH2_VRC_01.i_xClsLS <-> Channel 4/Input
//     PlcTask Inputs/GVL_VAC_VALVES.DREAM_ROUGH1_VRC_01.i_xOpnLS <-> Channel 1/Input
//     PlcTask Inputs/GVL_VAC_VALVES.DREAM_ROUGH2_VRC_01.i_xOpnLS <-> Channel 3/Input
//   lcls_plc_dream_vac Instance <-> Device 1 (EtherCAT)/R20_DRL_03_CX0_EK1200/R20_DRL_03_E15_EL1122/K4S8_DRL_04_EP1_EP4374-0002
//     PlcTask Inputs/GVL_VAC_GAUGES.DREAM_ROUGH1_GPI_02.i_iPRESS_R <-> AI Inputs Channel 1/Value
//     PlcTask Inputs/GVL_VAC_GAUGES.DREAM_ROUGH2_GPI_02.i_iPRESS_R <-> AI Inputs Channel 2/Value
//     PlcTask Outputs/GVL_VAC_VALVES.DREAM_ROUGH1_VFV_02.q_iRawPosition <-> AO Outputs Channel 3/Analog output
//     PlcTask Outputs/GVL_VAC_VALVES.DREAM_ROUGH2_VFV_02.q_iRawPosition <-> AO Outputs Channel 4/Analog output
//   lcls_plc_dream_vac Instance <-> Device 1 (EtherCAT)/R20_DRL_03_CX0_EK1200/R20_DRL_03_E15_EL1122/K4S8_DRL_04_EP2_EP4374-0002
//     PlcTask Inputs/GVL_VAC_GAUGES.DREAM_ROUGH2_GPI_03.i_iPRESS_R <-> AI Inputs Channel 1/Value
//     PlcTask Outputs/GVL_VAC_VALVES.DREAM_ROUGH2_VFV_03.q_iRawPosition <-> AO Outputs Channel 3/Analog output
//   lcls_plc_dream_vac Instance <-> Device 1 (EtherCAT)/R20_DRL_03_CX0_EK1200/R20_DRL_03_E15_EL1122/R03_DRL_01_EK1100/R03_DRL_01_E1_EL1004
//     PlcTask Inputs/GVL_VAC_GAUGES.DREAM_MC_GHC.i_xCH2_SEL <-> Channel 2/Input
//     PlcTask Inputs/GVL_VAC_GAUGES.DREAM_MC_GHC.i_xERR_CH1 <-> Channel 3/Input
//     PlcTask Inputs/GVL_VAC_GAUGES.DREAM_MC_GHC.i_xERR_CH2 <-> Channel 4/Input
//     PlcTask Inputs/GVL_VAC_GAUGES.DREAM_MC_GHC.i_xHV_ON <-> Channel 1/Input
//   lcls_plc_dream_vac Instance <-> Device 1 (EtherCAT)/R20_DRL_03_CX0_EK1200/R20_DRL_03_E15_EL1122/R03_DRL_01_EK1100/R03_DRL_01_E2_EL2624
//     PlcTask Outputs/GVL_VAC_GAUGES.DREAM_MC_GHC.q_xHV_DIS_CH1 <-> Channel 1/Output
//     PlcTask Outputs/GVL_VAC_GAUGES.DREAM_MC_GHC.q_xHV_DIS_CH2 <-> Channel 2/Output
//   lcls_plc_dream_vac Instance <-> Device 1 (EtherCAT)/R20_DRL_03_CX0_EK1200/R20_DRL_03_E15_EL1122/R03_DRL_01_EK1100/R03_DRL_01_E3_EL3174-0002
//     PlcTask Inputs/GVL_VAC_GAUGES.DREAM_MC_GHC.i_iPRESS_R_CH1 <-> AI Standard Channel 1/Value
//     PlcTask Inputs/GVL_VAC_GAUGES.DREAM_MC_GHC.i_iPRESS_R_CH2 <-> AI Standard Channel 2/Value
//   lcls_plc_dream_vac Instance <-> Device 1 (EtherCAT)/R20_DRL_03_CX0_EK1200/R20_DRL_03_E15_EL1122/WALL_E_PPL_01_EP1_EP4374-0002
//     PlcTask Inputs/GVL_VAC_GAUGES.DREAM_ROUGH1_GPI_01.i_iPRESS_R <-> AI Inputs Channel 1/Value
//     PlcTask Inputs/GVL_VAC_GAUGES.DREAM_ROUGH2_GPI_01.i_iPRESS_R <-> AI Inputs Channel 2/Value
//     PlcTask Outputs/GVL_VAC_VALVES.DREAM_ROUGH1_VFV_01.q_iRawPosition <-> AO Outputs Channel 3/Analog output
//     PlcTask Outputs/GVL_VAC_VALVES.DREAM_ROUGH2_VFV_01.q_iRawPosition <-> AO Outputs Channel 4/Analog output
//   lcls_plc_dream_vac Instance <-> Device 1 (EtherCAT)/R20_DRL_03_CX0_EK1200/R20_DRL_03_E15_EL1122/WALL_E_PPL_01_EP2_EP2338-0002
//     PlcTask Inputs/GVL_VAC_VALVES.DREAM_ROUGH1_VRC_10.i_xClsLS <-> Channel 2/Input
//     PlcTask Inputs/GVL_VAC_VALVES.DREAM_ROUGH1_VRC_10.i_xOpnLS <-> Channel 1/Input
//     PlcTask Outputs/GVL_VAC_VALVES.DREAM_ROUGH1_VRC_10.q_xOPN_DO <-> Channel 11/Output
//   lcls_plc_dream_vac Instance <-> Device 1 (EtherCAT)/R20_DRL_03_CX0_EK1200/R20_DRL_03_E4_EL1004
//     PlcTask Inputs/GVL_VAC_PUMPS.DREAM_DP2_PTM_01.i_xAtSpd <-> Channel 2/Input
//     PlcTask Inputs/GVL_VAC_PUMPS.DREAM_DP3_PTM_01.i_xAtSpd <-> Channel 4/Input
//     PlcTask Inputs/GVL_VAC_PUMPS.DREAM_DP2_PTM_01.i_xFaultNC <-> Channel 1/Input
//     PlcTask Inputs/GVL_VAC_PUMPS.DREAM_DP3_PTM_01.i_xFaultNC <-> Channel 3/Input
//   lcls_plc_dream_vac Instance <-> Device 1 (EtherCAT)/R20_DRL_03_CX0_EK1200/R20_DRL_03_E5_EL1004
//     PlcTask Inputs/GVL_VAC_PUMPS.DREAM_MC_PTM_01.i_xAtSpd <-> Channel 2/Input
//     PlcTask Inputs/GVL_VAC_PUMPS.DREAM_MC_PTM_02.i_xAtSpd <-> Channel 4/Input
//     PlcTask Inputs/GVL_VAC_PUMPS.DREAM_MC_PTM_01.i_xFaultNC <-> Channel 1/Input
//     PlcTask Inputs/GVL_VAC_PUMPS.DREAM_MC_PTM_02.i_xFaultNC <-> Channel 3/Input
//   lcls_plc_dream_vac Instance <-> Device 1 (EtherCAT)/R20_DRL_03_CX0_EK1200/R20_DRL_03_E7_EL2794
//     PlcTask Outputs/GVL_VAC_PUMPS.DREAM_DP2_PTM_01.q_RunDO <-> Channel 1/Output
//     PlcTask Outputs/GVL_VAC_PUMPS.DREAM_DP3_PTM_01.q_RunDO <-> Channel 3/Output
//     PlcTask Outputs/GVL_VAC_PUMPS.DREAM_MC_PTM_01.q_RunDO <-> Channel 2/Output
//     PlcTask Outputs/GVL_VAC_PUMPS.DREAM_MC_PTM_02.q_RunDO <-> Channel 4/Output
//   lcls_plc_dream_vac Instance <-> Device 1 (EtherCAT)/R20_DRL_03_CX0_EK1200/R20_DRL_03_E9_EL6001
//     Serial_COM Inputs/GVL_Serial_Com.stComIn_DREAM_DP2_PTM_01/D[0] <-> COM Inputs/Data In 0
//     Serial_COM Inputs/GVL_Serial_Com.stComIn_DREAM_DP2_PTM_01/D[10] <-> COM Inputs/Data In 10
//     Serial_COM Inputs/GVL_Serial_Com.stComIn_DREAM_DP2_PTM_01/D[11] <-> COM Inputs/Data In 11
//     Serial_COM Inputs/GVL_Serial_Com.stComIn_DREAM_DP2_PTM_01/D[12] <-> COM Inputs/Data In 12
//     Serial_COM Inputs/GVL_Serial_Com.stComIn_DREAM_DP2_PTM_01/D[13] <-> COM Inputs/Data In 13
//     Serial_COM Inputs/GVL_Serial_Com.stComIn_DREAM_DP2_PTM_01/D[14] <-> COM Inputs/Data In 14
//     Serial_COM Inputs/GVL_Serial_Com.stComIn_DREAM_DP2_PTM_01/D[15] <-> COM Inputs/Data In 15
//     Serial_COM Inputs/GVL_Serial_Com.stComIn_DREAM_DP2_PTM_01/D[16] <-> COM Inputs/Data In 16
//     Serial_COM Inputs/GVL_Serial_Com.stComIn_DREAM_DP2_PTM_01/D[17] <-> COM Inputs/Data In 17
//     Serial_COM Inputs/GVL_Serial_Com.stComIn_DREAM_DP2_PTM_01/D[18] <-> COM Inputs/Data In 18
//     Serial_COM Inputs/GVL_Serial_Com.stComIn_DREAM_DP2_PTM_01/D[19] <-> COM Inputs/Data In 19
//     Serial_COM Inputs/GVL_Serial_Com.stComIn_DREAM_DP2_PTM_01/D[1] <-> COM Inputs/Data In 1
//     Serial_COM Inputs/GVL_Serial_Com.stComIn_DREAM_DP2_PTM_01/D[20] <-> COM Inputs/Data In 20
//     Serial_COM Inputs/GVL_Serial_Com.stComIn_DREAM_DP2_PTM_01/D[21] <-> COM Inputs/Data In 21
//     Serial_COM Inputs/GVL_Serial_Com.stComIn_DREAM_DP2_PTM_01/D[2] <-> COM Inputs/Data In 2
//     Serial_COM Inputs/GVL_Serial_Com.stComIn_DREAM_DP2_PTM_01/D[3] <-> COM Inputs/Data In 3
//     Serial_COM Inputs/GVL_Serial_Com.stComIn_DREAM_DP2_PTM_01/D[4] <-> COM Inputs/Data In 4
//     Serial_COM Inputs/GVL_Serial_Com.stComIn_DREAM_DP2_PTM_01/D[5] <-> COM Inputs/Data In 5
//     Serial_COM Inputs/GVL_Serial_Com.stComIn_DREAM_DP2_PTM_01/D[6] <-> COM Inputs/Data In 6
//     Serial_COM Inputs/GVL_Serial_Com.stComIn_DREAM_DP2_PTM_01/D[7] <-> COM Inputs/Data In 7
//     Serial_COM Inputs/GVL_Serial_Com.stComIn_DREAM_DP2_PTM_01/D[8] <-> COM Inputs/Data In 8
//     Serial_COM Inputs/GVL_Serial_Com.stComIn_DREAM_DP2_PTM_01/D[9] <-> COM Inputs/Data In 9
//     Serial_COM Inputs/GVL_Serial_Com.stComIn_DREAM_DP2_PTM_01/Status <-> COM Inputs/Status
//     Serial_COM Outputs/GVL_Serial_Com.stComOut_DREAM_DP2_PTM_01/Ctrl <-> COM Outputs/Ctrl
//     Serial_COM Outputs/GVL_Serial_Com.stComOut_DREAM_DP2_PTM_01/D[0] <-> COM Outputs/Data Out 0
//     Serial_COM Outputs/GVL_Serial_Com.stComOut_DREAM_DP2_PTM_01/D[10] <-> COM Outputs/Data Out 10
//     Serial_COM Outputs/GVL_Serial_Com.stComOut_DREAM_DP2_PTM_01/D[11] <-> COM Outputs/Data Out 11
//     Serial_COM Outputs/GVL_Serial_Com.stComOut_DREAM_DP2_PTM_01/D[12] <-> COM Outputs/Data Out 12
//     Serial_COM Outputs/GVL_Serial_Com.stComOut_DREAM_DP2_PTM_01/D[13] <-> COM Outputs/Data Out 13
//     Serial_COM Outputs/GVL_Serial_Com.stComOut_DREAM_DP2_PTM_01/D[14] <-> COM Outputs/Data Out 14
//     Serial_COM Outputs/GVL_Serial_Com.stComOut_DREAM_DP2_PTM_01/D[15] <-> COM Outputs/Data Out 15
//     Serial_COM Outputs/GVL_Serial_Com.stComOut_DREAM_DP2_PTM_01/D[16] <-> COM Outputs/Data Out 16
//     Serial_COM Outputs/GVL_Serial_Com.stComOut_DREAM_DP2_PTM_01/D[17] <-> COM Outputs/Data Out 17
//     Serial_COM Outputs/GVL_Serial_Com.stComOut_DREAM_DP2_PTM_01/D[18] <-> COM Outputs/Data Out 18
//     Serial_COM Outputs/GVL_Serial_Com.stComOut_DREAM_DP2_PTM_01/D[19] <-> COM Outputs/Data Out 19
//     Serial_COM Outputs/GVL_Serial_Com.stComOut_DREAM_DP2_PTM_01/D[1] <-> COM Outputs/Data Out 1
//     Serial_COM Outputs/GVL_Serial_Com.stComOut_DREAM_DP2_PTM_01/D[20] <-> COM Outputs/Data Out 20
//     Serial_COM Outputs/GVL_Serial_Com.stComOut_DREAM_DP2_PTM_01/D[21] <-> COM Outputs/Data Out 21
//     Serial_COM Outputs/GVL_Serial_Com.stComOut_DREAM_DP2_PTM_01/D[2] <-> COM Outputs/Data Out 2
//     Serial_COM Outputs/GVL_Serial_Com.stComOut_DREAM_DP2_PTM_01/D[3] <-> COM Outputs/Data Out 3
//     Serial_COM Outputs/GVL_Serial_Com.stComOut_DREAM_DP2_PTM_01/D[4] <-> COM Outputs/Data Out 4
//     Serial_COM Outputs/GVL_Serial_Com.stComOut_DREAM_DP2_PTM_01/D[5] <-> COM Outputs/Data Out 5
//     Serial_COM Outputs/GVL_Serial_Com.stComOut_DREAM_DP2_PTM_01/D[6] <-> COM Outputs/Data Out 6
//     Serial_COM Outputs/GVL_Serial_Com.stComOut_DREAM_DP2_PTM_01/D[7] <-> COM Outputs/Data Out 7
//     Serial_COM Outputs/GVL_Serial_Com.stComOut_DREAM_DP2_PTM_01/D[8] <-> COM Outputs/Data Out 8
//     Serial_COM Outputs/GVL_Serial_Com.stComOut_DREAM_DP2_PTM_01/D[9] <-> COM Outputs/Data Out 9

CONFIGURATION lcls_plc_dream_vac
    RESOURCE PLC ON TwinCAT3
        TASK PlcTask(INTERVAL := T#10ms, PRIORITY := 20);
        TASK Serial_COM(INTERVAL := T#2ms, PRIORITY := 19);
        PROGRAM MAIN WITH PlcTask : MAIN;
        PROGRAM PRG_AUTOMATION WITH PlcTask : PRG_AUTOMATION;
        PROGRAM PRG_COM WITH Serial_COM : PRG_COM;
    END_RESOURCE
END_CONFIGURATION

// ---- DUTs/E_Op.TcDUT
TYPE E_Op :
(
    INIT := 0,  //Initialize system
    //IDLE := 1,  //State Machine IDLE, no operation
    STANDBY := 1, //Monitoring IF full system under vacuum
    PUMP_ALL := 2, //Full system pump down
    PUMP_NC := 3, //Only Nozzle chamber pump down
    AT_VACUUM := 4, //Monitor Vacuum status
    VENT_ALL := 5, //Vent full system
    VENT_NC := 6, //Vent nozzle chamber only
    VENT_MC_CAT := 7, //Vent Main Chamber + cather
    VENT_CAT := 8 //Vent cather only
);
END_TYPE

// ---- DUTs/E_OpStep.TcDUT
TYPE E_OpStep :
(
    IDLE := 0,
    START := 1,

    (* Vent MC and CAT System steps *)
    VMCAS_CLOSE_ISOLATION_VALVES,
    VMCAS_STOP_TURBO_PUMPS,
    VMCAS_CLOSE_ROUGH_VALVES,
    VMCAS_STOP_GAUGES,
    VMCAS_WAIT_FOR_TURBO_PUMPS_SPIN_DOWN,
    VMCAS_VENTING,
    VMCAS_FINISH
    (* Add new states for other procedures *)
);
END_TYPE

// ---- GVLs/GVL_Automation.TcGVL
VAR_GLOBAL
    // Execute flags for vacuum system operations
    {attribute 'pytmc' := '
        pv: PLC:DREAM:OPERATION
        io: io
    '}
    iq_eOperation : E_Op;

    {attribute 'pytmc' := '
        pv: PLC:DREAM:OPERATION:CANCEL
        io: io
    '}
    i_bCancel : BOOL;

    {attribute 'pytmc' := '
        pv: PLC:DREAM:OPERATION:RESET_ERROR
        io: io
    '}
    i_bResetError : BOOL;

    {attribute 'pytmc' := '
        pv: PLC:DREAM:OPERATION:BUSY
        io: i
        field: ZNAM NOT_BUSY
        field: ONAM BUSY
    '}
    q_bBusy : BOOL;

    {attribute 'pytmc' := '
        pv: PLC:DREAM:OPERATION:ERROR
        io: i
        field: ZNAM OK
        field: ONAM ERROR
        field: ZSV NO_ALARM
        field: OSV MAJOR
    '}
    q_bError : BOOL;

    {attribute 'pytmc' := '
        pv: PLC:DREAM:OPERATION:MESSAGE
        io: i
    '}
    q_sMessage : STRING(EPICS_STRING_SIZE);
END_VAR

// ---- GVLs/GVL_Constants.TcGVL
VAR_GLOBAL CONSTANT
    EPICS_STRING_SIZE : INT := 40;

    ATM_PRESS : REAL := 760.0; // Atmospheric pressure in Torr
    ATM_PRESS_INTERLOCK_SP : INT := 800; // Interlock pressure SP for valves
    ATM_PRESS_ERR_RNG : INT := 10; // Error range that is still considered atmospheric pressure // update while testing these values

    PTM_INTERLOCK_SP : REAL := 1E-2; // Turbo pumps interlock backing pressure SP
    VALVE_INTERLOCK_SP : REAL := 5E-3; // Roughing valve interlock pressure SP

    AT_VAC_SP : REAL := 1E-6; // Setpoint for at vacuum condition // update based on James and Jing input

    VALVE_TIMEOUT : TIME := T#10S; // How long system tries to open or close valve before failing
    TURBOS_NOT_RUNNING_TIMEOUT : TIME := T#10M; // How long to try turbo pumping before failing
    TURBOS_SPINDOWN_TIMEOUT : TIME := T#60M; // How long for turbos to spin down

    //Vent Valves
    VENTING_CYCLE : TIME := T#2M; // Increase open position every 2 min
    VFV_POSITION_STEP : INT := 1; // Position increase step
    ROUGH2_VFV_02_INITIAL_POSITION : INT := 50; // Initial postion in % for ROUGH2_VFV_02 valve
    ROUGH2_VFV_03_INITIAL_POSITION : INT := 40; // Initial postion in % for ROUGH2_VFV_03 valve
END_VAR

// ---- GVLs/GVL_FWM.TcGVL
//{attribute 'qualified_only'}
VAR_GLOBAL
    (*
    {attribute 'pytmc' := 'pv: DREAM:COIL'}
    {attribute 'TcLinkTo' := '.iRaw := TIIB[K4S8_DRL_03_E21_EL3052]^AI Standard Channel 1^Value'}
    fbDreamCoilFlowMeter : FB_FDQ_FlowMeter;
    *)

    {attribute 'TcLinkTo' := '.iRaw	:=	TIIB[K4S8_DRL_03_E21_EL3052]^AI Standard Channel 1^Value'}
    fbCoilFlowMeter : FB_AnalogInput := (iTermBits:=15, fTermMax:=60, fTermMin:=0);

    {attribute 'pytmc' := '
        pv: DREAM:COIL:FWM:VAL
        io: i
        field: EGU "lpm"
    '}
    fCoilCoolantFlowMeterRBV : LREAL;

    //Coil PS Current Monitoring
    {attribute 'TcLinkTo' := '.iRaw	:=	TIIB[K4S8_DRL_04_E16_EL3174-0002]^AI Standard Channel 4^Value'}
    fbCoilCurrentMonitoring : FB_AnalogInput := (iTermBits:=15, fTermMax:=310, fTermMin:=0);

    {attribute 'pytmc' := '
        pv: DREAM:COIL:CURRENT:VAL
        io: i
        field: EGU "A"
        field: PREC "2"
    '}
    fCoilCurrentRBV : LREAL;
END_VAR

// ---- GVLs/GVL_PLC_Interface.TcGVL
//{attribute 'qualified_only'}
VAR_GLOBAL
    (*ETHERCAT BRRIDGE COM STATUS*)
    //0: Other side is in OP state, >0: Error
    {attribute 'TcLinkTo' := 'TIIB[R20_DRL_03_E14_EL6695]^SYNC Inputs^TxPDO state'}
    bEcatBridge_TxPDO_state AT %I* :BOOL;

    //0: External device connectd, 1: External device not connected
    {attribute 'TcLinkTo' :=  'TIIB[R20_DRL_03_E14_EL6695]^SYNC Inputs^External device not connected'}
    bEcatBridge_External_device_not_connected AT %I* : BOOL;

    //0 = Data valid, 1 = Data invalid
    {attribute 'TcLinkTo' :=  'TIIB[R20_DRL_03_E14_EL6695]^WcState^WcStateIn'}
    bEcatBridge_WcState AT %I* : BOOL;

    (*Inputs from TMO Beamline*)
    {attribute 'TcLinkTo' :=  'TIIB[R20_DRL_03_E14_EL6695]^IO Inputs^HUTCH_PLC_NAME'}
    sHUTCH_PLC_NAME AT %I* : STRING(8);

    {attribute 'TcLinkTo' :=  'TIIB[R20_DRL_03_E14_EL6695]^IO Inputs^TMO_MR5K4_VWC_CLOSED_LS'}
    bTMO_MR5K4_VWC_CLOSED_LS AT %I* : BOOL;

    {attribute 'TcLinkTo' :=  'TIIB[R20_DRL_03_E14_EL6695]^IO Inputs^TMO_TM2K4_VWC_CLOSED_LS'}
    bTMO_TM2K4_VWC_CLOSED_LS AT %I* : BOOL;

    {attribute 'TcLinkTo' :=  'TIIB[R20_DRL_03_E14_EL6695]^IO Inputs^TMO_MR5K4_VWC_OPEN_LS'}
    bTMO_MR5K4_VWC_OPEN_LS AT %I* : BOOL;

    {attribute 'TcLinkTo' :=  'TIIB[R20_DRL_03_E14_EL6695]^IO Inputs^TMO_TM2K4_VWC_OPEN_LS'}
    bTMO_TM2K4_VWC_OPEN_LS AT %I* : BOOL;

    (*Outputs to TMO Beamline PLC*)
    {attribute 'TcLinkTo' :=   'TIIB[R20_DRL_03_E14_EL6695]^IO Outputs^ENDSTATION_PLC_NAME'}
    sENDSTATION_PLC_NAME AT %Q* : STRING(8):= 'DREAM';

    {attribute 'TcLinkTo' :=  'TIIB[R20_DRL_03_E14_EL6695]^IO Outputs^DREAM_HV_SAFETY_ENABLE'}
    bDREAM_HV_SAFETY_ENABLE AT %Q* : BOOL;

    {attribute 'TcLInkTo' :=  'TIIB[R20_DRL_03_E14_EL6695]^IO Outputs^DREAM_TURBOS_ALL_AtSpd'}
    {attribute 'pytmc' := '
        pv: PLC:DREAM:VAC:TURBOS_ALL_ATSPD
        io: i
    '}
    bDREAM_TURBOS_ALL_AtSpd AT %Q* : BOOL;

    {attribute 'TcLinkTo' :=  'TIIB[R20_DRL_03_E14_EL6695]^IO Outputs^DREAM_MAIN_xAT_VAC'}
    bDREAM_MAIN_xAT_VAC AT %Q* : BOOL;

    {attribute 'TcLInkTo' :=  'TIIB[R20_DRL_03_E14_EL6695]^IO Outputs^DREAM_MAIN_xPRESS_OK'}
    bDREAM_MAIN_xPRESS_OK AT %Q* : BOOL;

    {attribute 'TcLINKTo' :=  'TIIB[R20_DRL_03_E14_EL6695]^IO Outputs^DREAM_MAIN_rPRESS'}
    fDREAM_MAIN_rPRESS AT %Q* : REAL;

    {attribute 'TcLinkTo' :=  'TIIB[R20_DRL_03_E14_EL6695]^IO Outputs^CLOSE_TMO_MR5K4_VWC'}
    bCLOSE_TMO_MR5K4_VWC AT %Q* : BOOL;

    {attribute 'TcLinkTo' :=  'TIIB[R20_DRL_03_E14_EL6695]^IO Outputs^CLOSE_TMO_TM2K4_VWC'}
    bCLOSE_TMO_TM2K4_VWC AT %Q* : BOOL;

    (*ISEG HV Crate Safety Loop*)
    {attribute 'TcLInkTo' :=  'TIIB[K4S8_DRL_04_E14_EL2624]^Channel 4^Output'}
    {attribute 'pytmc' := '
        pv: TMO:PLC:DREAM:VAC:HV_SAFETY_ENABLE
        io:i
    '}
    bHVSafteyLoopEnable AT %Q* : BOOL := FALSE; (*When Enables the High voltage Saftey loop is closed and HV can start.*)

    (*Interlock output to control COIL PS*)
    {attribute 'TcLInkTo' :=  'TIIB[K4S8_DRL_04_E14_EL2624]^Channel 3^Output'}
    {attribute 'pytmc' := '
        pv: PLC:DREAM:COIL_PS:ILK
        io: i
    '}
    bCoilPS_ILK AT %Q* : BOOL := FALSE;

    //Ethercat interface with DREAM motion PLC

     (*ETHERCAT BRRIDGE COM STATUS*)
    //0: Other side is in OP state, >0: Error
    {attribute 'TcLinkTo' := 'TIIB[R20_DRL_03_E15_EL1122]^SYNC Inputs^TxPDO state'}
    bMotEcatBridge_TxPDO_state AT %I* :BOOL;

    //0: External device connectd, 1: External device not connected
    {attribute 'TcLinkTo' :=  'TIIB[R20_DRL_03_E14_EL6695]^SYNC Inputs^External device not connected'}
    bMotEcatBridge_External_device_not_connected AT %I* : BOOL;

    //0 = Data valid, 1 = Data invalid
    {attribute 'TcLinkTo' :=  'TIIB[R20_DRL_03_E15_EL1122]^WcState^WcStateIn'}
    bMotEcatBridge_WcState AT %I* : BOOL;

    (*Inputs from DREAM Motion*)
    //{attribute 'TcLinkTo' :=  'TIIB[R20_DRL_03_E14_EL6695]^IO Inputs^HUTCH_PLC_NAME'}
    //sMOT_PLC_NAME AT %I* : STRING(8);

    {attribute 'TcLinkTo' :=  'TIIB[R20_DRL_03_E15_EL1122]^IO Outputs^xDREAM_GNZ_Y_OUT'}
    xDREAM_GNZ_Y_OUT AT %I* : BOOL;

    {attribute 'TcLinkTo' :=  'TIIB[R20_DRL_03_E15_EL1122]IO Outputs^xDREAM_GNZ_Y_Ext_OUT'}
    xDREAM_GNZ_Y_Ext_OUT AT %I* : BOOL;

    (*Outputs to DREAM Motion*)
    {attribute 'TcLinkTo' :=  'TIIB[R20_DRL_03_E15_EL1122]^IO Inputs^bDREAM_VRC_DP1_OPENED_LS'}
    bDREAM_VRC_DP1_OPENED_LS AT %Q* : BOOL;

END_VAR

// ---- GVLs/GVL_Serial_Com.TcGVL
//{attribute 'qualified_only'}
VAR_GLOBAL
    //COMM FUNCTION
    SerialRXBuffer_DREAM_NC_PTM_01     : ComBuffer;
    SerialTXBuffer_DREAM_NC_PTM_01     : ComBuffer;
    SerialRXBuffer_DREAM_NC_PTM_02     : ComBuffer;
    SerialTXBuffer_DREAM_NC_PTM_02     : ComBuffer;
    SerialRXBuffer_DREAM_DP1_PTM_01    : ComBuffer;
    SerialTXBuffer_DREAM_DP1_PTM_01    : ComBuffer;
    SerialRXBuffer_DREAM_DP2_PTM_01    : ComBuffer;
    SerialTXBuffer_DREAM_DP2_PTM_01    : ComBuffer;
    SerialRXBuffer_DREAM_DP3_PTM_01    : ComBuffer;
    SerialTXBuffer_DREAM_DP3_PTM_01    : ComBuffer;
    SerialRXBuffer_DREAM_MC_PTM_01     : ComBuffer;
    SerialTXBuffer_DREAM_MC_PTM_01     : ComBuffer;
    SerialRXBuffer_DREAM_MC_PTM_02     : ComBuffer;
    SerialTXBuffer_DREAM_MC_PTM_02     : ComBuffer;
    SerialRXBuffer_DREAM_CAT1_PTM_01   : ComBuffer;
    SerialTXBuffer_DREAM_CAT1_PTM_01   : ComBuffer;
    SerialRXBuffer_DREAM_CAT2_PTM_01   : ComBuffer;
    SerialTXBuffer_DREAM_CAT2_PTM_01   : ComBuffer;
    SerialRXBuffer_DREAM_ROUGH2_PTM_01 : ComBuffer;
    SerialTXBuffer_DREAM_ROUGH2_PTM_01 : ComBuffer;
    SerialRXBuffer_DREAM_ROUGH2_PTM_02 : ComBuffer;
    SerialTXBuffer_DREAM_ROUGH2_PTM_02 : ComBuffer;

    //Serial Terminal
    fbSerialLineControl_DREAM_NC_PTM_01     : SerialLineControl;
    fbSerialLineControl_DREAM_NC_PTM_02     : SerialLineControl;
    fbSerialLineControl_DREAM_DP1_PTM_01    : SerialLineControl;
    fbSerialLineControl_DREAM_DP2_PTM_01    : SerialLineControl;
    fbSerialLineControl_DREAM_DP3_PTM_01    : SerialLineControl;
    fbSerialLineControl_DREAM_MC_PTM_01     : SerialLineControl;
    fbSerialLineControl_DREAM_MC_PTM_02     : SerialLineControl;
    fbSerialLineControl_DREAM_CAT1_PTM_01   : SerialLineControl;
    fbSerialLineControl_DREAM_CAT2_PTM_01   : SerialLineControl;
    fbSerialLineControl_DREAM_ROUGH2_PTM_01 : SerialLineControl;
    fbSerialLineControl_DREAM_ROUGH2_PTM_02 : SerialLineControl;

    //SERIAL IO
    {attribute	'TcLinkTo'	:=	'.Status:=TIIB[K4S8_DRL_03_E12_EL6021]^COM TxPDO-Map Inputs^Status;
                                 .D[0]:=TIIB[K4S8_DRL_03_E12_EL6021]^COM TxPDO-Map Inputs^Data In 0;
                                 .D[1]:=TIIB[K4S8_DRL_03_E12_EL6021]^COM TxPDO-Map Inputs^Data In 1;
                                 .D[2]:=TIIB[K4S8_DRL_03_E12_EL6021]^COM TxPDO-Map Inputs^Data In 2;
                                 .D[3]:=TIIB[K4S8_DRL_03_E12_EL6021]^COM TxPDO-Map Inputs^Data In 3;
                                 .D[4]:=TIIB[K4S8_DRL_03_E12_EL6021]^COM TxPDO-Map Inputs^Data In 4;
                                 .D[5]:=TIIB[K4S8_DRL_03_E12_EL6021]^COM TxPDO-Map Inputs^Data In 5;
                                 .D[6]:=TIIB[K4S8_DRL_03_E12_EL6021]^COM TxPDO-Map Inputs^Data In 6;
                                 .D[7]:=TIIB[K4S8_DRL_03_E12_EL6021]^COM TxPDO-Map Inputs^Data In 7;
                                 .D[8]:=TIIB[K4S8_DRL_03_E12_EL6021]^COM TxPDO-Map Inputs^Data In 8;
                                 .D[9]:=TIIB[K4S8_DRL_03_E12_EL6021]^COM TxPDO-Map Inputs^Data In 9;
                                 .D[10]:=TIIB[K4S8_DRL_03_E12_EL6021]^COM TxPDO-Map Inputs^Data In 10;
                                 .D[11]:=TIIB[K4S8_DRL_03_E12_EL6021]^COM TxPDO-Map Inputs^Data In 11;
                                 .D[12]:=TIIB[K4S8_DRL_03_E12_EL6021]^COM TxPDO-Map Inputs^Data In 12;
                                 .D[13]:=TIIB[K4S8_DRL_03_E12_EL6021]^COM TxPDO-Map Inputs^Data In 13;
                                 .D[14]:=TIIB[K4S8_DRL_03_E12_EL6021]^COM TxPDO-Map Inputs^Data In 14;
                                 .D[15]:=TIIB[K4S8_DRL_03_E12_EL6021]^COM TxPDO-Map Inputs^Data In 15;
                                 .D[16]:=TIIB[K4S8_DRL_03_E12_EL6021]^COM TxPDO-Map Inputs^Data In 16;
                                 .D[17]:=TIIB[K4S8_DRL_03_E12_EL6021]^COM TxPDO-Map Inputs^Data In 17;
                                 .D[18]:=TIIB[K4S8_DRL_03_E12_EL6021]^COM TxPDO-Map Inputs^Data In 18;
                                 .D[19]:=TIIB[K4S8_DRL_03_E12_EL6021]^COM TxPDO-Map Inputs^Data In 19;
                                 .D[20]:=TIIB[K4S8_DRL_03_E12_EL6021]^COM TxPDO-Map Inputs^Data In 20;
                                 .D[21]:=TIIB[K4S8_DRL_03_E12_EL6021]^COM TxPDO-Map Inputs^Data In 21
    '}
    stComIn_DREAM_NC_PTM_01 AT %I* : EL6inData22B;

    {attribute 'TcLinkTo'	:=	'.Ctrl:=TIIB[K4S8_DRL_03_E12_EL6021]^COM RxPDO-Map Outputs^Ctrl;
                                 .D[0]:=TIIB[K4S8_DRL_03_E12_EL6021]^COM RxPDO-Map Outputs^Data Out 0;
                                 .D[1]:=TIIB[K4S8_DRL_03_E12_EL6021]^COM RxPDO-Map Outputs^Data Out 1;
                                 .D[2]:=TIIB[K4S8_DRL_03_E12_EL6021]^COM RxPDO-Map Outputs^Data Out 2;
                                 .D[3]:=TIIB[K4S8_DRL_03_E12_EL6021]^COM RxPDO-Map Outputs^Data Out 3;
                                 .D[4]:=TIIB[K4S8_DRL_03_E12_EL6021]^COM RxPDO-Map Outputs^Data Out 4;
                                 .D[5]:=TIIB[K4S8_DRL_03_E12_EL6021]^COM RxPDO-Map Outputs^Data Out 5;
                                 .D[6]:=TIIB[K4S8_DRL_03_E12_EL6021]^COM RxPDO-Map Outputs^Data Out 6;
                                 .D[7]:=TIIB[K4S8_DRL_03_E12_EL6021]^COM RxPDO-Map Outputs^Data Out 7;
                                 .D[8]:=TIIB[K4S8_DRL_03_E12_EL6021]^COM RxPDO-Map Outputs^Data Out 8;
                                 .D[9]:=TIIB[K4S8_DRL_03_E12_EL6021]^COM RxPDO-Map Outputs^Data Out 9;
                                 .D[10]:=TIIB[K4S8_DRL_03_E12_EL6021]^COM RxPDO-Map Outputs^Data Out 10;
                                 .D[11]:=TIIB[K4S8_DRL_03_E12_EL6021]^COM RxPDO-Map Outputs^Data Out 11;
                                 .D[12]:=TIIB[K4S8_DRL_03_E12_EL6021]^COM RxPDO-Map Outputs^Data Out 12;
                                 .D[13]:=TIIB[K4S8_DRL_03_E12_EL6021]^COM RxPDO-Map Outputs^Data Out 13;
                                 .D[14]:=TIIB[K4S8_DRL_03_E12_EL6021]^COM RxPDO-Map Outputs^Data Out 14;
                                 .D[15]:=TIIB[K4S8_DRL_03_E12_EL6021]^COM RxPDO-Map Outputs^Data Out 15;
                                 .D[16]:=TIIB[K4S8_DRL_03_E12_EL6021]^COM RxPDO-Map Outputs^Data Out 16;
                                 .D[17]:=TIIB[K4S8_DRL_03_E12_EL6021]^COM RxPDO-Map Outputs^Data Out 17;
                                 .D[18]:=TIIB[K4S8_DRL_03_E12_EL6021]^COM RxPDO-Map Outputs^Data Out 18;
                                 .D[19]:=TIIB[K4S8_DRL_03_E12_EL6021]^COM RxPDO-Map Outputs^Data Out 19;
                                 .D[20]:=TIIB[K4S8_DRL_03_E12_EL6021]^COM RxPDO-Map Outputs^Data Out 20;
                                 .D[21]:=TIIB[K4S8_DRL_03_E12_EL6021]^COM RxPDO-Map Outputs^Data Out 21
    '}
    stComOut_DREAM_NC_PTM_01 AT %Q* : EL6outData22B;

    {attribute	'TcLinkTo'	:=	'.Status:=TIIB[K4S8_DRL_03_E15_EL6021]^COM TxPDO-Map Inputs^Status;
                                 .D[0]:=TIIB[K4S8_DRL_03_E15_EL6021]^COM TxPDO-Map Inputs^Data In 0;
                                 .D[1]:=TIIB[K4S8_DRL_03_E15_EL6021]^COM TxPDO-Map Inputs^Data In 1;
                                 .D[2]:=TIIB[K4S8_DRL_03_E15_EL6021]^COM TxPDO-Map Inputs^Data In 2;
                                 .D[3]:=TIIB[K4S8_DRL_03_E15_EL6021]^COM TxPDO-Map Inputs^Data In 3;
                                 .D[4]:=TIIB[K4S8_DRL_03_E15_EL6021]^COM TxPDO-Map Inputs^Data In 4;
                                 .D[5]:=TIIB[K4S8_DRL_03_E15_EL6021]^COM TxPDO-Map Inputs^Data In 5;
                                 .D[6]:=TIIB[K4S8_DRL_03_E15_EL6021]^COM TxPDO-Map Inputs^Data In 6;
                                 .D[7]:=TIIB[K4S8_DRL_03_E15_EL6021]^COM TxPDO-Map Inputs^Data In 7;
                                 .D[8]:=TIIB[K4S8_DRL_03_E15_EL6021]^COM TxPDO-Map Inputs^Data In 8;
                                 .D[9]:=TIIB[K4S8_DRL_03_E15_EL6021]^COM TxPDO-Map Inputs^Data In 9;
                                 .D[10]:=TIIB[K4S8_DRL_03_E15_EL6021]^COM TxPDO-Map Inputs^Data In 10;
                                 .D[11]:=TIIB[K4S8_DRL_03_E15_EL6021]^COM TxPDO-Map Inputs^Data In 11;
                                 .D[12]:=TIIB[K4S8_DRL_03_E15_EL6021]^COM TxPDO-Map Inputs^Data In 12;
                                 .D[13]:=TIIB[K4S8_DRL_03_E15_EL6021]^COM TxPDO-Map Inputs^Data In 13;
                                 .D[14]:=TIIB[K4S8_DRL_03_E15_EL6021]^COM TxPDO-Map Inputs^Data In 14;
                                 .D[15]:=TIIB[K4S8_DRL_03_E15_EL6021]^COM TxPDO-Map Inputs^Data In 15;
                                 .D[16]:=TIIB[K4S8_DRL_03_E15_EL6021]^COM TxPDO-Map Inputs^Data In 16;
                                 .D[17]:=TIIB[K4S8_DRL_03_E15_EL6021]^COM TxPDO-Map Inputs^Data In 17;
                                 .D[18]:=TIIB[K4S8_DRL_03_E15_EL6021]^COM TxPDO-Map Inputs^Data In 18;
                                 .D[19]:=TIIB[K4S8_DRL_03_E15_EL6021]^COM TxPDO-Map Inputs^Data In 19;
                                 .D[20]:=TIIB[K4S8_DRL_03_E15_EL6021]^COM TxPDO-Map Inputs^Data In 20;
                                 .D[21]:=TIIB[K4S8_DRL_03_E15_EL6021]^COM TxPDO-Map Inputs^Data In 21
    '}
    stComIn_DREAM_NC_PTM_02 AT %I* : EL6inData22B;

    {attribute 'TcLinkTo'	:=	'.Ctrl:=TIIB[K4S8_DRL_03_E15_EL6021]^COM RxPDO-Map Outputs^Ctrl;
                                 .D[0]:=TIIB[K4S8_DRL_03_E15_EL6021]^COM RxPDO-Map Outputs^Data Out 0;
                                 .D[1]:=TIIB[K4S8_DRL_03_E15_EL6021]^COM RxPDO-Map Outputs^Data Out 1;
                                 .D[2]:=TIIB[K4S8_DRL_03_E15_EL6021]^COM RxPDO-Map Outputs^Data Out 2;
                                 .D[3]:=TIIB[K4S8_DRL_03_E15_EL6021]^COM RxPDO-Map Outputs^Data Out 3;
                                 .D[4]:=TIIB[K4S8_DRL_03_E15_EL6021]^COM RxPDO-Map Outputs^Data Out 4;
                                 .D[5]:=TIIB[K4S8_DRL_03_E15_EL6021]^COM RxPDO-Map Outputs^Data Out 5;
                                 .D[6]:=TIIB[K4S8_DRL_03_E15_EL6021]^COM RxPDO-Map Outputs^Data Out 6;
                                 .D[7]:=TIIB[K4S8_DRL_03_E15_EL6021]^COM RxPDO-Map Outputs^Data Out 7;
                                 .D[8]:=TIIB[K4S8_DRL_03_E15_EL6021]^COM RxPDO-Map Outputs^Data Out 8;
                                 .D[9]:=TIIB[K4S8_DRL_03_E15_EL6021]^COM RxPDO-Map Outputs^Data Out 9;
                                 .D[10]:=TIIB[K4S8_DRL_03_E15_EL6021]^COM RxPDO-Map Outputs^Data Out 10;
                                 .D[11]:=TIIB[K4S8_DRL_03_E15_EL6021]^COM RxPDO-Map Outputs^Data Out 11;
                                 .D[12]:=TIIB[K4S8_DRL_03_E15_EL6021]^COM RxPDO-Map Outputs^Data Out 12;
                                 .D[13]:=TIIB[K4S8_DRL_03_E15_EL6021]^COM RxPDO-Map Outputs^Data Out 13;
                                 .D[14]:=TIIB[K4S8_DRL_03_E15_EL6021]^COM RxPDO-Map Outputs^Data Out 14;
                                 .D[15]:=TIIB[K4S8_DRL_03_E15_EL6021]^COM RxPDO-Map Outputs^Data Out 15;
                                 .D[16]:=TIIB[K4S8_DRL_03_E15_EL6021]^COM RxPDO-Map Outputs^Data Out 16;
                                 .D[17]:=TIIB[K4S8_DRL_03_E15_EL6021]^COM RxPDO-Map Outputs^Data Out 17;
                                 .D[18]:=TIIB[K4S8_DRL_03_E15_EL6021]^COM RxPDO-Map Outputs^Data Out 18;
                                 .D[19]:=TIIB[K4S8_DRL_03_E15_EL6021]^COM RxPDO-Map Outputs^Data Out 19;
                                 .D[20]:=TIIB[K4S8_DRL_03_E15_EL6021]^COM RxPDO-Map Outputs^Data Out 20;
                                 .D[21]:=TIIB[K4S8_DRL_03_E15_EL6021]^COM RxPDO-Map Outputs^Data Out 21
    '}
    stComOut_DREAM_NC_PTM_02 AT %Q* : EL6outData22B;

